# B&R Automation Studio project IP001 (part 2)

#### FValve.st
```iecst
(* ЗАДВИЖКА *)
FUNCTION_BLOCK FValve
	IF r0.14 THEN
		r0.14 := 0;
		Failures := 0;
	END_IF
	IF Failures = 0 THEN					//Сброс таймаутов
		TimeoutC := 0;
		TimeoutO := 0;
		OpenNoAllow := 0;
		CloseNoAllow := 0;
		NoOpenNoAllow := 0;
		NoCloseNoAllow := 0;
	END_IF;
	(* разбираем регистр команд *)
	IF r0.0 THEN
		Open := 1;	r0.0 := 0;
	END_IF;
	IF r0.1 THEN
		Close := 1;	r0.1 := 0;
	END_IF;
	IF r0.2 THEN
		Stop := 1; r0.2 := 0;
	END_IF

	Block	:= r0.3;
	Auto	:= r0.5;
	Imitation := r0.13;

	IF PAZ THEN
		Open := 0;
		Close := 0;
		Stop := 0;
	END_IF
	(* Блокировка неактуальных команд *)
	IF Block THEN
		Open	:= 0;
		Close	:= 0;
		Stop	:= 0;
	END_IF;

	IF Open AND Opened THEN
		Open := 0;
	END_IF;
	IF Close AND Closed THEN
		Close := 0;
	END_IF;
	(*	режим иммитации	*)
	IF NOT Imitation THEN
		Opened	:= OpenedDI;
		Closed	:= ClosedDI;
	ELSE
		IF Opening AND T.ET > T#2s THEN Opened	:= 1; END_IF;
		IF Closing AND T.ET > T#2s THEN Closed	:= 1; END_IF;
	END_IF;
	(* команды *)
	IF Open THEN									// команда ОТКРЫТЬ
		Closing	:= 0;
		Closed	:= 0;
		CloseDO	:= 0;
		Open	:= 0;
		Opening	:= 1;
		OpenDO	:= 1 AND NOT Imitation AND NOT PAZ;
		T(IN	:= 1);
	END_IF;
	IF Opening AND Opened THEN						// Открылась
		Opening	:= 0;
		OpenDO	:= 0;
		OpenDIOld := OpenedDI;
		StopDO	:= 1  AND NOT Imitation;
		T(IN	:= 0);
	END_IF;
	IF Opening AND T.Q THEN							// НЕ Открылась
		Opening	:= 0;
		OpenDO	:= 0;
		T(IN	:= 0);
		TimeoutO:= 1;
	END_IF;

	IF Close THEN											// команда ЗАКРЫТЬ
		Opening	:= 0;
		Opened	:= 0;
		OpenDO	:= 0;
		Close	:= 0;
		Closing	:= 1;
		CloseDO	:= 1 AND NOT Imitation AND NOT PAZ;
		T(IN	:= 1);
	END_IF;
	IF Closing AND Closed THEN								// Закрылась
		Closing	:= 0;
		CloseDO	:= 0;
		CloseDIOld := ClosedDI;
		T(IN	:= 0);
		StopDO	:= 1;
	END_IF;
	IF Closing AND T.Q THEN									// НЕ Закрылась
		Closing	:= 0;
		CloseDO	:= 0;
		T(IN	:= 0);
		TimeoutC:= 1;
	END_IF;

	IF Stop	THEN											// Команда СТОП
		Stop	:= 0;
		Opening	:= 0;
		Closing	:= 0;
		OpenDO	:= 0;
		CloseDO	:= 0;
		T.IN	:= 0;
		StopDO	:= 1 AND NOT Imitation AND NOT PAZ;
	END_IF;

	IF StopPresent AND TSignal.Q THEN						// DO сигналы делаем 1 сек если есть сигнал StopDO
		OpenDO	:= 0;
		CloseDO	:= 0;
		StopDO	:= 0;
	END_IF;

	IF Block THEN											// при блокеровке обнуляем выходные сигналы
		OpenDO	:= 0;
		CloseDO	:= 0;
		StopDO	:= 0;
	END_IF;
	// Блокировка по ПАЗ или команда РЕМОНТ
	IF PAZ OR r0.10 THEN
		Opening	:= 0;
		Closing	:= 0;
		OpenDO	:= 0;
		CloseDO	:= 0;
		T.IN	:= 0;
		StopDO	:= 0;
	END_IF;
	(* Самопроизвольное открытие/закрытие *)
	IF Opening AND NOT ClosedDI THEN
		CloseDIOld := 0;
	END_IF;
	IF Closing AND NOT OpenedDI THEN
		OpenDIOld := 0;
	END_IF;
	IF OpenedDI AND NOT OpenDIOld THEN
		OpenDIOld := OpenedDI;
		OpenNoAllow := 1;
	END_IF;
	IF ClosedDI AND NOT CloseDIOld THEN
		CloseDIOld := ClosedDI;
		CloseNoAllow := 1;
	END_IF;
	IF NOT OpenedDI AND OpenDIOld THEN
		OpenDIOld := OpenedDI;
		NoOpenNoAllow := 1;
	END_IF;
	IF NOT ClosedDI AND CloseDIOld THEN
		CloseDIOld := ClosedDI;
		NoCloseNoAllow := 1;
	END_IF;
	(* Утечки *)
	// LeakTON(IN := LeakDI, PT := DINT_TO_TIME(LeakageTimer));
	// вызов таймера хода (30 сек по дефолту)
	T(PT := DINT_TO_TIME(FullTimerInterval));
	TSignal(IN := CloseDO OR OpenDO OR StopDO);
	(* Регистр состояний *)
	r1.0	:= NOT Block;									//  программный 1:может управл с контроллера; 0:только слежение за состоянием, без управл
	r1.1	:= TimeoutC OR TimeoutO;									// контроль (наличие) протечки
	r1.2	:= Auto;										// Режим АВТОМАТИЧЕСКИЙ
	r1.3 	:= NOT Auto;									// Режим РУЧНОЙ
	r1.4	:= Opening;										//  открывается
	r1.5	:= Closing;										//  закрывается
	r1.6	:= Opened;										//	открыта
	r1.7	:= Closed;										//	закрыта
	r1.8	:= (NOT OpenedDI AND NOT ClosedDI)AND NOT(OpenDO OR CloseDO);					//	в промежуточном положении

	//r1.10	:= AlarmDI;										// аварийное отключение или сработала муфта
	//r1.11 связи с интерфейсной задвижкой (0-нет связи, 1-есть связь)
	r1.12	:= NOT Block;									//	Работоспособен:= (если программный или имитационный, и если не блокирован)
	r1.13	:= NOT Block AND NOT PAZ AND NOT r0.10;		//	Готова
	r1.14	:= PAZ;											// задвижка под управлением ПАЗ
	(* Регистор аварий *)
	Failures.0	:= TimeoutC OR TimeoutO;					// Не открылась/закрылась за время T.PT
	// превышение времени схода с концевого выключателя
	Failures.2	:= TimeoutC OR TimeoutO;					// превышение времени полного хода вала
	// 3
	Failures.4	:= TimeoutO;								//	не выполнение команды открыть
	Failures.5	:= TimeoutC;								//	не выполнение команды закрыть
	// 6
	//7	сработала электрозащита
	//8	невыполнение команды останова
	//9	Сработал моментный выключатель открытия
	//10	Сработал моментный выключатель закрытия
	//11	Привод перегрелся
	Failures.12 := OpenNoAllow;
	Failures.13 := CloseNoAllow;
	Failures.14 := NoOpenNoAllow;
	Failures.15 := NoCloseNoAllow;

END_FUNCTION_BLOCK
```

#### FAI.st
```iecst
(* Обработка AI *)
FUNCTION_BLOCK FAI
	ImitationEn := 	RegCmd.1;
	HiEnabled := 	RegCmd.4;
	HiHiEnabled :=	RegCmd.5;
	LoEnabled := 	RegCmd.6;
	LoLoEnabled := 	RegCmd.7;
	Scale := HiScale - LoScale;	//шкала
	CASE ChannelType OF
		0:
			Current := RAW*20.0/32767.0;
			Value := RAW*((Scale+Scale/4)/32767.0) + (LoScale - Scale/4.0);
			Invalid := (ChannelOverflow OR ChannelUnderflow OR Current <= 3.2) AND NOT ImitationEn;// КЗ/обрыв
		1:
			Current := RAW*16.0/32767.0 + 4.0;
			Value := RAW*(Scale /32767.0) + LoScale;
			Invalid := (ChannelOverflow OR ChannelUnderflow OR Current <= 3.2) AND NOT ImitationEn;// КЗ/обрыв
		2:
			Current := RAW*22.0/32767.0;
			Value := RAW*(Scale+Scale/4)/32767.0 - Scale/4;
			Invalid := (ChannelOverflow OR ChannelUnderflow) AND NOT ImitationEn;// КЗ/обрыв
		3:
			Current := 0;
			Value := MbValue;
			Invalid := (ChannelOverflow OR ChannelUnderflow) AND NOT ImitationEn;// КЗ/обрыв
	END_CASE
	//Value := (Current - 4.0) / 16.0 * Scale + LoScale;
	IF ImitationEn THEN
		Value := Replace_Value;	// подстановочное
	ELSE
		IF Value < LoScale THEN
			Value := LoScale;
		END_IF;
		IF Value > HiScale THEN
			Value := HiScale;
		END_IF;
	END_IF;

	(* Аварии *)
	IF LoLoAlarm AND (Value >= (LoLoLimit + Scale*(Hyst/100.0)))OR  NOT LoLoEnabled OR Invalid THEN
		LoLoAlarm := 0;
	END_IF;
	IF NOT LoLoAlarm AND (Value < LoLoLimit)AND LoLoEnabled AND NOT Invalid THEN
		LoLoAlarm := 1;
	END_IF;
	IF LoAlarm AND (Value >= (LoLimit + Scale*(Hyst/100.0)))OR  NOT LoEnabled OR Invalid THEN
		LoAlarm := 0;
	END_IF;
	IF NOT LoAlarm AND (Value < LoLimit)AND LoEnabled AND NOT Invalid THEN
		LoAlarm := 1;
	END_IF;
	IF HiAlarm AND (Value <= (HiLimit - Scale*(Hyst/100.0)))OR  NOT HiEnabled OR Invalid THEN
		HiAlarm := 0;
	END_IF;
	IF NOT HiAlarm AND (Value > HiLimit)AND HiEnabled AND NOT Invalid THEN
		HiAlarm := 1;
	END_IF;
	IF HiHiAlarm AND (Value <= (HiHiLimit - Scale*(Hyst/100.0)))OR  NOT HiHiEnabled OR Invalid THEN
		HiHiAlarm := 0;
	END_IF;
	IF NOT HiHiAlarm AND (Value > HiHiLimit )AND HiHiEnabled AND NOT Invalid THEN
		HiHiAlarm := 1;
	END_IF;

	Color := 1;
	IF LoAlarm OR HiAlarm THEN
		Color := 2;
	END_IF
	IF LoLoAlarm OR HiHiAlarm THEN
		Color := 3;
	END_IF
	IF Invalid THEN
		Color := 4;
	END_IF

	RegStatus.0	:= Invalid;						//Сигнал достоверен (=FALSE) или нет (=TRUE)
	RegStatus.1	:= HiAlarm;						//Значение выше чем предупредительная уставка "HiLimit"
	RegStatus.2	:= HiHiAlarm;					//Значение выше чем аварийная уставка "HiHiLimit"
	RegStatus.3	:= LoAlarm;						//Значение ниже чем предупредительная уставка "LoLimit"
	RegStatus.4	:= LoLoAlarm;					//Значение ниже чем аварийная уставка "LoLoLimit"
	RegStatus.5 := ImitationEn;					//Включена имитация

END_FUNCTION_BLOCK
```

#### FDI.st
```iecst
(*Обработка дискретных входов*)
FUNCTION_BLOCK FDI
	Out := ((In XOR Inv) AND NOT MaskEn)OR(MaskEn AND Mask);
END_FUNCTION_BLOCK
```

#### FDO.st
```iecst
(*Обработка дискретных выходов*)
FUNCTION_BLOCK FDO
	Out	:= ((In	XOR Inv)	AND NOT MaskEn)	OR(MaskEn		AND Mask);
END_FUNCTION_BLOCK
```

#### FAO.st
```iecst
(* Обработка AO *)
FUNCTION_BLOCK FAO

	Scale := HiScale - LoScale;										//шкала
	IF ImitationEn THEN
		Value := Replace_Value;	  									// подстановочное
	END_IF

	RAW := REAL_TO_INT((Value-LoScale)*(32767.0)/(HiScale-LoScale));		// Величину в АЦП канала
	Current := RAW*16.0/32767.0+4.0;										// АЦП в ТОК

	(* Аварии *)
	IF LoLoAlarm AND (Value > (LoLoLimit + Scale/200.0))OR  NOT LoLoEnabled OR Invalid THEN
		LoLoAlarm := 0;
	END_IF;
	IF NOT LoLoAlarm AND (Value < (LoLoLimit - Scale/200.0))AND LoLoEnabled AND NOT Invalid THEN
		LoLoAlarm := 1;
	END_IF;
	IF LoAlarm AND (Value > (LoLimit + Scale/200.0))OR  NOT LoEnabled OR Invalid THEN
		LoAlarm := 0;
	END_IF;
	IF NOT LoAlarm AND (Value < (LoLimit - Scale/200.0))AND LoEnabled AND NOT Invalid THEN
		LoAlarm := 1;
	END_IF;
	IF HiAlarm AND (Value < (HiLimit - Scale/200.0))OR  NOT HiEnabled OR Invalid THEN
		HiAlarm := 0;
	END_IF;
	IF NOT HiAlarm AND (Value > (HiLimit + Scale/200.0))AND HiEnabled AND NOT Invalid THEN
		HiAlarm := 1;
	END_IF;
	IF HiHiAlarm AND (Value < (HiHiLimit - Scale/200.0))OR  NOT HiHiEnabled OR Invalid THEN
		HiHiAlarm := 0;
	END_IF;
	IF NOT HiHiAlarm AND (Value > (HiHiLimit + Scale/200.0))AND HiHiEnabled AND NOT Invalid THEN
		HiHiAlarm := 1;
	END_IF;
END_FUNCTION_BLOCK
```

#### FPIDreg_r.st
```iecst
FUNCTION_BLOCK FPIDreg_r
	IF AlOpen THEN mode := 3; END_IF
	IF AlClose THEN mode := 4; END_IF
	IF enable THEN
		status := 0;
		MTBasicsPID_0.Invert := invert;
		MTBasicsPID_0.MinOut := Y_min;
		MTBasicsPID_0.MaxOut := Y_max;
		MTBasicsPID_0.SetValue := X_set;
		MTBasicsPID_0.ActValue := X;
		IF (MTBasicsPID_0.PIDParameters.Gain <> Gain) OR (MTBasicsPID_0.PIDParameters.IntegrationTime <> IntegrationTime)
			OR (MTBasicsPID_0.PIDParameters.DerivativeTime <> DerivativeTime)OR (MTBasicsPID_0.PIDParameters.FilterTime <> FilterTime) THEN
			MTBasicsPID_0.PIDParameters.Gain := Gain;
			MTBasicsPID_0.PIDParameters.IntegrationTime := IntegrationTime;
			MTBasicsPID_0.PIDParameters.DerivativeTime := DerivativeTime;
			MTBasicsPID_0.PIDParameters.FilterTime := FilterTime;
			MTBasicsPID_0.Update := TRUE;
		ELSE MTBasicsPID_0.Update := FALSE;
		END_IF
		CASE mode OF
			0://выключен
				MTBasicsPID_0.Enable := FALSE;
			1://автоматический режим
				MTBasicsPID_0.Enable := TRUE;
				MTBasicsPID_0.EnableTracking := FALSE;
				IF MTBasicsPID_0.IntegrationPartPresetValue <> MTBasicsPID_0.TrackingValue THEN
					MTBasicsPID_0.IntegrationPartPresetValue := MTBasicsPID_0.TrackingValue;
				END_IF
				IF NOT MTBasicsPID_0.EnableTracking AND MTBasicsPID_0.TrackingActive THEN
					MTBasicsPID_0.SetIntegrationPart := TRUE;
				ELSE 	MTBasicsPID_0.SetIntegrationPart := FALSE;
				END_IF
			2://ручной режим
				MTBasicsPID_0.Enable := TRUE;
				MTBasicsPID_0.EnableTracking := TRUE;
				MTBasicsPID_0.TrackingValue := Y_man;
			3://в ручном на макс
				MTBasicsPID_0.Enable := TRUE;
				MTBasicsPID_0.EnableTracking := TRUE;
				MTBasicsPID_0.TrackingValue := MTBasicsPID_0.MaxOut;
			4://в ручном на мин
				MTBasicsPID_0.Enable := TRUE;
				MTBasicsPID_0.EnableTracking := TRUE;
				MTBasicsPID_0.TrackingValue := MTBasicsPID_0.MinOut;
			ELSE
				mode := 2;
		END_CASE

		MTBasicsPID_0();
		Y_out := MTBasicsPID_0.Out;
		status := MTBasicsPID_0.StatusID;
	END_IF
END_FUNCTION_BLOCK
```

#### FMotor.st
```iecst
FUNCTION_BLOCK FMotor
	IF Block THEN
		Start	:= 0;
		Stop	:= 1;
	END_IF
	Started_old := Started;
	Stopped_old := Stopped;
	IF Block AND Started THEN
		Status.5 := TRUE;
	END_IF
	IF Status.5 AND Reset AND Stopped THEN
		Status.5 := FALSE;
	END_IF
	//Имитация
	IF NOT Imitation THEN
		Started := RunDI;
		Stopped := NOT RunDI;
	ELSE
		IF Start THEN Started := 1; Stopped := 0; END_IF
		IF Stop THEN Started := 0; Stopped := 1; END_IF
	END_IF
	IF Start AND Started THEN				// Блокировка неактуальных команд
		Start := 0;
	END_IF
	IF Stop AND Stopped THEN
		Stop := 0;
	END_IF
	IF Reset THEN							// Таймаут Сбрс
		Reset	:= 0;
		Timeout	:= 0;
	END_IF
	IF Start THEN							// СТАРТ
		Start	:= 0;
		StartDO	:= 1;
		T.IN := 1;
	END_IF
	IF Stop THEN							// СТОП
		Stop	:= 0;
		StopDO	:= 1;
		T.IN := 1;
	END_IF
	IF (StartDO OR StopDO) AND T.Q THEN		// Таймаут
		StartDO	:= 0;
		StopDO	:= 0;
		T.IN	:= 0;
		Timeout	:= 1;
	END_IF
	IF StartDO AND RunDI THEN				// Стартовал
		StartDO := 0;
		T.IN	:= 0;
		Timeout	:= 0;
	END_IF

	IF StopDO AND NOT RunDI THEN			// Остановился
		StopDO := 0;
		T.IN	:= 0;
		Timeout	:= 0;
	END_IF
	T(IN := T.IN,	PT := T#3s00ms);
	MH(Run := Started,Reset := ResetMH);
	ResetMH := 0;
	MotoHours := MH.Counter;
	Status.0	:= Started;
	Status.1 	:= Stopped;
	Status.2 	:= Block;
	Status.3	:= Timeout;
	Status.4	:= Timeout;

END_FUNCTION_BLOCK
```

#### PassportValve.st
```iecst
(* TODO: Add your comment here *)
FUNCTION_BLOCK PassportValve
	IF is_first THEN
		is_first := 0;
		cmdOpen := Gate_buf.r0.0;
		cmdClose := Gate_buf.r0.1;
		cmdBlck := Gate_buf.r0.3;
		cmdAuto := Gate_buf.r0.5;
		cmdImit := Gate_buf.r0.13;
		statePLC_control := Gate_buf.r1.0;
		stateLeak := Gate_buf.r1.1;
		stateAuto := Gate_buf.r1.2;
		stateManu := Gate_buf.r1.3;
		stateOpening := Gate_buf.r1.4;
		stateClosing := Gate_buf.r1.5;
		stateOpened := Gate_buf.r1.6;
		stateClosed := Gate_buf.r1.7;
		statePAZ := Gate_buf.r1.14;
		failTimeout := Gate_buf.Failures.0 OR Gate_buf.Failures.2;
		failTimeoutO := Gate_buf.Failures.4;
		failTimeoutC := Gate_buf.Failures.5;
		timePT := Gate_buf.FullTimerInterval/1000;
	ELSE
		Gate_buf.r0.0 := cmdOpen;
		Gate_buf.r0.1 := cmdClose;
		Gate_buf.r0.3 := cmdBlck;
		Gate_buf.r0.5 := cmdAuto;
		Gate_buf.r0.13 := cmdImit;
		statePLC_control := Gate_buf.r1.0;
		stateLeak := Gate_buf.r1.1;
		stateAuto := Gate_buf.r1.2;
		stateManu := Gate_buf.r1.3;
		stateOpening := Gate_buf.r1.4;
		stateClosing := Gate_buf.r1.5;
		stateOpened := Gate_buf.r1.6;
		stateClosed := Gate_buf.r1.7;
		statePAZ := Gate_buf.r1.14;
		failTimeout := Gate_buf.Failures.0 OR Gate_buf.Failures.2;
		failTimeoutO := Gate_buf.Failures.4;
		failTimeoutC := Gate_buf.Failures.5;
		Gate_buf.FullTimerInterval := timePT*1000;
		IF cmdResetAlarms THEN
			Gate_buf.r0.14 := 1;
			cmdResetAlarms := 0;
		END_IF
	END_IF
END_FUNCTION_BLOCK
```

#### PassportAI.st
```iecst
FUNCTION_BLOCK PassportAI
	IF is_first THEN
		index1_old	:= index1;
		index2_old	:= index2;
		is_first 	:= 0;
		LoScale 	:= AI_buf.LoScale;
		HiScale 	:= AI_buf.HiScale;
		HiLimit 	:= AI_buf.HiLimit;
		HiHiLimit 	:= AI_buf.HiHiLimit;
		LoLimit 	:= AI_buf.LoLimit;
		LoLoLimit 	:= AI_buf.LoLoLimit;
		current 	:= AI_buf.Current;
		Value 		:= AI_buf.Value;
		ImitVal 	:= AI_buf.Replace_Value;
		cmdImit 	:= AI_buf.ImitationEn;
		cmdHiEn 	:= AI_buf.HiEnabled;
		cmdHiHiEn 	:= AI_buf.HiHiEnabled;
		cmdLoEn 	:= AI_buf.LoEnabled;
		cmdLoLoEn 	:= AI_buf.LoLoEnabled;
		stateInvalid:= AI_buf.Invalid;
		stateHi 	:= AI_buf.HiAlarm;
		stateHiHi 	:= AI_buf.HiHiAlarm;
		stateLo 	:= AI_buf.LoAlarm;
		stateLoLo 	:= AI_buf.LoLoAlarm;

	ELSE
		IF index1_old = index1 AND index2_old = index2 THEN
			current := AI_buf.Current;
			Value := AI_buf.Value;
			stateInvalid:= AI_buf.Invalid;
			stateHi 	:= AI_buf.HiAlarm;
			stateHiHi 	:= AI_buf.HiHiAlarm;
			stateLo 	:= AI_buf.LoAlarm;
			stateLoLo 	:= AI_buf.LoLoAlarm;
			AI_buf.LoScale := LoScale;
			AI_buf.HiScale := HiScale;
			AI_buf.HiLimit := HiLimit;
			AI_buf.HiHiLimit := HiHiLimit;
			AI_buf.LoLimit := LoLimit;
			AI_buf.LoLoLimit := LoLoLimit;
			AI_buf.Replace_Value := ImitVal;
			AI_buf.ImitationEn := cmdImit;
			AI_buf.HiEnabled := cmdHiEn;
			AI_buf.HiHiEnabled := cmdHiHiEn;
			AI_buf.LoEnabled := cmdLoEn;
			AI_buf.LoLoEnabled := cmdLoLoEn;
		ELSE is_first := 1;
		END_IF
	END_IF

END_FUNCTION_BLOCK
```

#### FDISKRreg_r.st
```iecst
(* Дискретный регулятор *)
FUNCTION_BLOCK FDISKRreg_r
	IF enable THEN
		IF invert THEN //регулятор ПОСЛЕ СЕБЯ
			IF X < X_set_low 	THEN OnDO := TRUE; OffDO := FALSE; END_IF
			IF X > X_set_high THEN OnDO := FALSE; OffDO := TRUE; END_IF
		ELSE			//регулятор ДО СЕБЯ
			IF X > X_set_high THEN OnDO := TRUE; OffDO := FALSE; END_IF
			IF X < X_set_low 	THEN OnDO := FALSE; OffDO := TRUE; END_IF
		END_IF
	ELSE OnDO := FALSE; OffDO := TRUE;
	END_IF
END_FUNCTION_BLOCK
```

#### UVP_TCP.st
```iecst
(* UVP_TCP *)
FUNCTION_BLOCK UVP_TCP
	CASE step OF
		0://чтение текущего времени УВП(+маска описанных трубопроводов)
			req_3x (enable := TRUE,pStation := pPort,startAddress :=1800,nrRegisters :=SIZEOF(UVP_Data.Time)/2 ,pData := ADR(UVP_Data.Time),dataSize :=SIZEOF(UVP_Data.Time));
			IF req_3x.status <> ERR_FUB_BUSY THEN
				step := 1;
			END_IF
			state := req_3x.status;
		1://чтение порядка байт
			req_3x (enable := TRUE,pStation := pPort,startAddress :=100,nrRegisters :=SIZEOF(UVP_Data.Byte_order)/2 ,pData := ADR(UVP_Data.Byte_order),dataSize :=SIZEOF(UVP_Data.Byte_order));
			IF req_3x.status <> ERR_FUB_BUSY THEN
				step := 2;
			END_IF
			state := req_3x.status;
		2://запись порядка байт,если он отличается от заданного(#2301)
			IF UVP_Data.Byte_order <> UVP_Data.Byte_order_new THEN
				req_6x (enable := TRUE,pStation := pPort,startAddress :=100,value := UVP_Data.Byte_order_new);
				IF req_6x.status <> ERR_FUB_BUSY THEN
					step := 3;
				END_IF
				state := req_6x.status;
			ELSE step := 3;
			END_IF
		3://чтение текущих параметров трубопровода(за один проход CASE один трубопровод)
			WHILE ((curTP <= 15) AND ((UVP_Data.Time.TPs AND SHL(1,curTP)) = 0)) DO
				curTP := curTP + 1;
			END_WHILE
			IF curTP > 15 THEN curTP := 0; END_IF
			IF ((UVP_Data.Time.TPs AND SHL(1,curTP))<>0) THEN
				req_4x(enable := TRUE,pStation := pPort,startAddress := 2000+(curTP*100), nrRegisters := SIZEOF(UVP_Data.LineCurrent[curTP+1])/2,pData := ADR(UVP_Data.LineCurrent[curTP+1]),dataSize :=SIZEOF(UVP_Data.LineCurrent[curTP+1]));
				IF req_4x.status <> ERR_FUB_BUSY THEN
					step := 4;
				END_IF
				state := req_4x.status;
			ELSE step := 4;
			END_IF
			//чтение текущих архивов(за один проход CASE один трубопровод)
		4:	IF ((UVP_Data.Time.TPs AND SHL(1,curTP))<>0) THEN
				req_4x(enable := TRUE,pStation := pPort,startAddress := 2000+(curTP*100)+60, nrRegisters := SIZEOF(UVP_Data.Prev_hour[curTP+1])/2,pData := ADR(UVP_Data.Prev_hour[curTP+1]),dataSize :=SIZEOF(UVP_Data.Prev_hour[curTP+1]));
				IF req_4x.status <> ERR_FUB_BUSY THEN
					step := 5;
				END_IF
				state := req_4x.status;
			ELSE step := 5;
			END_IF
			//чтение текущих архивов(за один проход CASE один трубопровод)
		5:	IF ((UVP_Data.Time.TPs AND SHL(1,curTP))<>0) THEN
				req_4x (enable := TRUE,pStation := pPort,startAddress := 2000+(curTP*100)+80, nrRegisters := SIZEOF(UVP_Data.Prev_day[curTP+1])/2,pData := ADR(UVP_Data.Prev_day[curTP+1]),dataSize :=SIZEOF(UVP_Data.Prev_day[curTP+1]));
				IF req_4x.status <> ERR_FUB_BUSY THEN
					curTP := curTP + 1;
					step := 6;
				END_IF
				state := req_4x.status;
			ELSE step := 6;
			END_IF
		6:  //синхронизация времени  с NTP сервером(в конфиге контроллера включен сервер)
			//IP адрес контроллера задан младшим словом вперед,т.к. порядяок байт #2301
			IF UVP_Data.synchrooo THEN
				UVP_Data.synchrooo := FALSE;
				UVP_Data.NTP.IPAddr1 := UVP_Data.NTP.IpAddress3*256 + UVP_Data.NTP.IpAddress4;
				UVP_Data.NTP.IPAddr2 := UVP_Data.NTP.IpAddress1*256 + UVP_Data.NTP.IpAddress2;
				UVP_Data.NTP.cmd := 24680;
				req_16x(enable := TRUE,pStation := pPort, startAddress := 1005, nrRegisters := SIZEOF(UVP_Data.NTP)/2,pData:=ADR(UVP_Data.NTP),dataSize := SIZEOF(UVP_Data.NTP));
				IF req_16x.status <> ERR_FUB_BUSY THEN
					step := 7;
				END_IF
				state := req_16x.status;
			ELSE step := 7;
			END_IF
		7://чтение текущего статуса синхронизации времени
			req_3x (enable := TRUE,pStation := pPort, startAddress := 1005, nrRegisters := (SIZEOF(UVP_Data.NTP)-4)/2,pData:=ADR(UVP_Data.NTP),dataSize := SIZEOF(UVP_Data.NTP)-4);
			IF req_3x.status <> ERR_FUB_BUSY THEN
				step := 8;
			END_IF
			state := req_3x.status;
		8:
			req_3x (enable := TRUE,pStation := pPort, startAddress := 1008, nrRegisters := SIZEOF(UVP_Data.DeltaTime)/2,pData:=ADR(UVP_Data.DeltaTime),dataSize := SIZEOF(UVP_Data.DeltaTime));
			IF req_3x.status <> ERR_FUB_BUSY THEN
				step := 9;
			END_IF
			state := req_3x.status;
		9://чтение компонентного состава газовой смеси МР-113
			IF UVP_Data.read_gas_comp THEN
				req_3x(enable := TRUE,pStation := pPort, startAddress := 1100, nrRegisters := SIZEOF(UVP_Data.MR_113)/2,pData:=ADR(UVP_Data.MR_113),dataSize := SIZEOF(UVP_Data.MR_113));
				IF req_3x.status  <> ERR_FUB_BUSY THEN
					UVP_Data.MR_113_new := UVP_Data.MR_113;
					UVP_Data.read_gas_comp := FALSE;
					step := 10;
				END_IF
				state := req_3x.status;
			ELSE step := 10;
			END_IF
		10://запись компонентного состава газовой смеси МР-113
			IF UVP_Data.write_gas_comp THEN
				req_16x(enable := TRUE, pStation := pPort, startAddress := 1100, nrRegisters := SIZEOF(UVP_Data.MR_113_new)/2,pData:=ADR(UVP_Data.MR_113_new),dataSize := SIZEOF(UVP_Data.MR_113_new));
				IF req_16x.status <> ERR_FUB_BUSY THEN
					UVP_Data.write_gas_comp := FALSE;
					step := 0;
				END_IF
				state := req_16x.status;
			ELSE step := 0;
			END_IF
	END_CASE;

	IF state = 34201 THEN
			status := state;
			Timeout_T (IN := TRUE, PT := T#5000ms);
			IF Timeout_T.Q THEN
				step := step + 1;
				Timeout_T (IN := FALSE, PT := T#5000ms);
		END_IF
	ELSE status := 0;
	END_IF

	IF step > 10 THEN step := 0; END_IF
END_FUNCTION_BLOCK
```

#### FMHCounter.st
```iecst
(* FMHCounter *)
FUNCTION_BLOCK FMHCounter
	T(IN := Run, PT :=  UINT_TO_TIME(Tik*1000));
	IF T.Q THEN
		Counter := Counter + (Tik/3600.00);
		T(IN := FALSE);
	END_IF
	IF Reset THEN Counter := 0; END_IF
END_FUNCTION_BLOCK
```

#### FTorch.st
```iecst
(* Torch *)
FUNCTION_BLOCK FTorch
	Timer_vent(PT := UINT_TO_TIME(Time_vent*1000));
	Timer_firing(PT := UINT_TO_TIME(Time_firing*1000));
	Timer_stabiliz(PT := UINT_TO_TIME(Time_stabiliz*1000));
	Timer_spark_off(PT := UINT_TO_TIME(Time_spark_off*1000));
	Timer_spark_on(PT := UINT_TO_TIME(Time_spark_on*1000));
	Timer_after_alarm(PT := UINT_TO_TIME(Time_after_alarm*1000));

	IF Stop THEN
		Timer_vent.IN := FALSE;
		Timer_firing.IN := FALSE;
		Timer_stabiliz.IN := FALSE;
		Timer_spark_off.IN := FALSE;
		Timer_spark_on.IN := FALSE;
		Timer_after_alarm.IN := FALSE;
		Do_Valve := FALSE;
		Do_Spark := FALSE;
		Do_Lamp_P_Zapal_low := FALSE;
		Do_Lamp_FireON := FALSE;
		Do_Lamp_Alarm := FALSE;
		step := 0;
		Stop := FALSE;
	END_IF
	Do_Lamp_Alarm := USINT_TO_BOOL(Alarm);
	Do_Lamp_FireON := Di_Fire;
	IF NOT Mode_Manual THEN
		CASE step OF
			0://Начальное состояние(ГОТОВНОСТЬ К ПУСКУ)
				IF Di_Fire THEN Warning_2 := TRUE;
				ELSE Warning_2 := FALSE; END_IF;
				IF Di_P_gas_low THEN Warning_1 := TRUE;
				ELSE Warning_1 := FALSE; END_IF;
				IF Start AND NOT Di_Fire AND NOT Di_P_gas_low THEN
					Start := FALSE;
					step := 1;
					Alarm := 0;
					firing_count := 0;
				END_IF;
			1:// ВЕНТИЛЯЦИЯ
				IF NOT Di_P_gas_low THEN
					Do_Valve := TRUE;
					Timer_vent.IN := TRUE;
					IF Timer_vent.Q THEN
						Timer_vent.IN := FALSE;
						step := 2;
					END_IF;
				ELSE
					Do_Lamp_P_Zapal_low := TRUE;
					Do_Valve := FALSE;
					Timer_vent.IN := FALSE;
					step := 0;
					Alarm := 1;//Падение давления во время вентиляции
				END_IF;
			2://РОЗЖИГ
				IF NOT Di_P_gas_low THEN
					Timer_firing.IN := TRUE;
					Timer_spark_on.IN := NOT Timer_spark_off.Q;
					Timer_spark_off.IN := Timer_spark_on.Q;
					Do_Spark := NOT Timer_spark_on.Q;
					IF Di_Fire THEN
						Timer_firing.IN := FALSE;
						Timer_spark_on.IN := FALSE;
						Timer_spark_off.IN := FALSE;
						Do_Spark :=FALSE;
						step := 4;
					END_IF;
					IF Timer_firing.Q THEN
						Timer_firing.IN := FALSE;
						Timer_spark_on.IN := FALSE;
						Timer_spark_off.IN := FALSE;
						Do_Spark :=FALSE;
						step := 3;
					END_IF;
				ELSE
					Do_Lamp_P_Zapal_low := TRUE;
					Timer_firing.IN := FALSE;
					Timer_spark_on.IN := FALSE;
					Timer_spark_off.IN := FALSE;
					Do_Spark :=FALSE;
					Do_Valve := FALSE;
					step := 0;
					Alarm := 2;//Падение давления во время розжига
				END_IF

			3://СТАБИЛИЗАЦИЯ
				IF NOT Di_P_gas_low THEN
					Timer_stabiliz.IN := TRUE;
					IF Di_Fire THEN
						Timer_stabiliz.IN := FALSE;
						step := 4;
						Alarm := 0;
					END_IF;
					IF Timer_stabiliz.Q THEN
						Timer_stabiliz.IN := FALSE;
						step := 5;
						Alarm := 3; //Нет розжига
					END_IF;
				ELSE
					Timer_stabiliz.IN := FALSE;
					Do_Lamp_P_Zapal_low := TRUE;
					Do_Valve := FALSE;
					step := 0;
					Alarm := 4;//Падение давления во время стабилизации
				END_IF
			4://ГОРЕНИЕ
				IF Di_P_gas_low THEN
					Alarm := 6;//Падение давления во время горения
					step := 5;
					Do_Lamp_P_Zapal_low := TRUE;
				END_IF
				IF NOT Di_Fire THEN
					Alarm := 7; //Срыв пламени
					firing_count := firing_count + 1;
					IF firing_count > 3 THEN
						step := 0;
					ELSE
						step := 2;
					END_IF
				END_IF
			5://АВАРИЯ
				Do_Valve := FALSE;
				Timer_after_alarm.IN := TRUE;
				IF Timer_after_alarm.Q THEN
					Timer_after_alarm.IN := FALSE;
					step := 0;
				END_IF
		END_CASE
	END_IF
END_FUNCTION_BLOCK
```

#### ABAK_TCP.st
```iecst
(* ABAK_MB_TCP *)
FUNCTION_BLOCK ABAK_TCP
	CASE step OF
		0:
		1:
		2:
		3:
		4:
	END_CASE
END_FUNCTION_BLOCK
```

#### FSwitch.st
```iecst
(* Switch *)
FUNCTION_BLOCK FSwitch
	IF Block THEN
		Start_1	:= 0;
		Start_2	:= 0;
		Stop	:= 1;
	END_IF
	IF Block_1 THEN
		Start_1 := 0;
	END_IF
	IF Block_2 THEN
		Start_2 := 0;
	END_IF
	IF Block_Stop THEN
		Stop := 0;
	END_IF
	//Имитация
	IF NOT Imitation THEN
		Started_1 := RunDI_1;
		Started_2 := RunDI_2;
		Stopped := NOT (RunDI_1 OR RunDI_2);
	ELSE
		IF Start_1 THEN Started_1 := 1; Started_2 := 0; Stopped := 0; END_IF
		IF Start_2 THEN Started_2 := 1; Started_1 := 0; Stopped := 0; END_IF
		IF Stop THEN Started_1 := 0; Started_2 := 0; Stopped := 1; END_IF
	END_IF

	IF Start_1 AND Started_1 THEN				// Блокировка неактуальных команд
		Start_1 := 0;
	END_IF
	IF Start_2 AND Started_2 THEN				// Блокировка неактуальных команд
		Start_2 := 0;
	END_IF
	IF Stop AND Stopped THEN
		Stop := 0;
	END_IF
	IF Reset THEN							// Таймаут Сбрс
		Reset	:= 0;
		Timeout	:= 0;
	END_IF
	IF Start_1 THEN							// СТАРТ
		Start_1	:= 0;
		Starting_1 := 1;
		Stop := 1;
	END_IF
	IF Start_2 THEN							// СТАРТ
		Start_2	:= 0;
		Starting_2 := 1;
		Stop := 1;
	END_IF
	IF Starting_1 AND Stopped THEN
		Starting_1 := 0;
		StartDO_1 := 1;
		T.IN := 1;
	END_IF
	IF Starting_2 AND Stopped THEN
		Starting_2 := 0;
		StartDO_2 := 1;
		T.IN := 1;
	END_IF
	IF Stop THEN							// СТОП
		Stop	:= 0;
		StopDO	:= 1;
		T.IN := 1;
	END_IF
	IF (StartDO_1 OR StartDO_2 OR StopDO) AND T.Q THEN		// Таймаут
		StartDO_1	:= 0;
		StartDO_2	:= 0;
		StopDO	:= 0;
		T.IN	:= 0;
		Timeout	:= 1;
	END_IF
	IF StartDO_1 AND RunDI_1 THEN				// Стартовал
		StartDO_1 := 0;
		T.IN	:= 0;
		Timeout	:= 0;
	END_IF
	IF StartDO_2 AND RunDI_2 THEN				// Стартовал
		StartDO_2 := 0;
		T.IN	:= 0;
		Timeout	:= 0;
	END_IF
	IF StopDO AND NOT RunDI_1 AND NOT RunDI_2 THEN			// Остановился
		StopDO := 0;
		T.IN	:= 0;
		Timeout	:= 0;
	END_IF
	T(IN := T.IN,	PT := T#3s00ms);

	Status.0	:= Started_1;
	Status.1	:= Started_2;
	Status.2 	:= Stopped;
	Status.3	:= Timeout;
	Status.4 	:= Block_1;
	Status.5 	:= Block_2;
	Status.6  	:= Block_Stop;

END_FUNCTION_BLOCK
```

#### fCmdCOM.st
```iecst
(* MBRTU Comm to ATV *)
FUNCTION_BLOCK fCmdCOM
	MBMCmd_0.ident := ident;
	MBMCmd_0.mfc := cmd;
	MBMCmd_0.node := node;
	MBMCmd_0.offset := offset;
	MBMCmd_0.len := length;
	MBMCmd_0.data := pData;
	MBMCmd_0(enable := TRUE);
	status := MBMCmd_0.status;
END_FUNCTION_BLOCK
```

#### fOpenCOM.st
```iecst
(*  *)
FUNCTION_BLOCK fOpenCOM
	IF enable THEN
		MBMOpen_0(enable := TRUE, pDevice := Device, pMode := Mode, pConfig := Config, timeout := 1500 );
		status := MBMOpen_0.status;
		ident := MBMOpen_0.ident;
		enable := FALSE;
	END_IF
END_FUNCTION_BLOCK
```

#### fCloseCOM.st
```iecst
(*  *)
FUNCTION_BLOCK fCloseCOM
	IF enable THEN
		MBMClose_0.ident := ident;
		MBMClose_0(enable := TRUE);
		status := MBMClose_0.status;
		enable := FALSE;
	END_IF
END_FUNCTION_BLOCK
```

#### FAlarm.st
```iecst
(* Alarm with delay *)
FUNCTION_BLOCK FAlarm
	Result := IN AND EN;
	IF Ack AND (Result = 0) THEN
		Timer(IN := FALSE);
		OUT := FALSE;
		OUT_int := Result;
	END_IF

	Timer(IN := UINT_TO_BOOL(Result), PT := UINT_TO_TIME(Delay*1000));
	IF Timer.Q THEN
		OUT := TRUE;
		OUT_int := Result;
	END_IF
END_FUNCTION_BLOCK
```

#### UVP_RTU.st
```iecst
(* UVP over RTU *)
FUNCTION_BLOCK UVP_RTU
	CASE step OF
			0://чтение текущего времени УВП(+маска описанных трубопроводов)
				req_3x (enable := TRUE,pStation := pPort,startAddress :=1800,nrRegisters :=SIZEOF(UVP_Data.Time)/2 ,pData := ADR(UVP_Data.Time),dataSize :=SIZEOF(UVP_Data.Time));
				IF req_3x.status <> ERR_FUB_BUSY THEN
					step := 1;
				END_IF
				state := req_3x.status;
			1://чтение порядка байт
				req_3x (enable := TRUE,pStation := pPort,startAddress :=100,nrRegisters :=SIZEOF(UVP_Data.Byte_order)/2 ,pData := ADR(UVP_Data.Byte_order),dataSize :=SIZEOF(UVP_Data.Byte_order));
				IF req_3x.status <> ERR_FUB_BUSY THEN
					step := 2;
				END_IF
				state := req_3x.status;
			2://запись порядка байт,если он отличается от заданного(#2301)
				IF UVP_Data.Byte_order <> UVP_Data.Byte_order_new THEN
					req_6x (enable := TRUE,pStation := pPort,startAddress :=100,pData := ADR(UVP_Data.Byte_order_new));
					IF req_6x.status <> ERR_FUB_BUSY THEN
						step := 3;
					END_IF
					state := req_6x.status;
				ELSE step := 3;
				END_IF
			3://чтение текущих параметров трубопровода(за один проход CASE один трубопровод)
				WHILE ((curTP <= 15) AND ((UVP_Data.Time.TPs AND SHL(1,curTP)) = 0)) DO
					curTP := curTP + 1;
				END_WHILE
				IF curTP > 15 THEN curTP := 0; END_IF
				IF ((UVP_Data.Time.TPs AND SHL(1,curTP))<>0) THEN
					req_4x(enable := TRUE,pStation := pPort,startAddress := 2000+(curTP*100), nrRegisters := SIZEOF(UVP_Data.LineCurrent[curTP+1])/2,pData := ADR(UVP_Data.LineCurrent[curTP+1]),dataSize :=SIZEOF(UVP_Data.LineCurrent[curTP+1]));
					IF req_4x.status <> ERR_FUB_BUSY THEN
						step := 4;
					END_IF
					state := req_4x.status;
				ELSE step := 4;
				END_IF
				//чтение текущих архивов(за один проход CASE один трубопровод)
			4:	IF ((UVP_Data.Time.TPs AND SHL(1,curTP))<>0) THEN
					req_4x(enable := TRUE,pStation := pPort,startAddress := 2000+(curTP*100)+60, nrRegisters := SIZEOF(UVP_Data.Prev_hour[curTP+1])/2,pData := ADR(UVP_Data.Prev_hour[curTP+1]),dataSize :=SIZEOF(UVP_Data.Prev_hour[curTP+1]));
					IF req_4x.status <> ERR_FUB_BUSY THEN
						step := 5;
					END_IF
					state := req_4x.status;
				ELSE step := 5;
				END_IF
				//чтение текущих архивов(за один проход CASE один трубопровод)
			5:	IF ((UVP_Data.Time.TPs AND SHL(1,curTP))<>0) THEN
					req_4x (enable := TRUE,pStation := pPort,startAddress := 2000+(curTP*100)+80, nrRegisters := SIZEOF(UVP_Data.Prev_day[curTP+1])/2,pData := ADR(UVP_Data.Prev_day[curTP+1]),dataSize :=SIZEOF(UVP_Data.Prev_day[curTP+1]));
					IF req_4x.status <> ERR_FUB_BUSY THEN
						curTP := curTP + 1;
						step := 6;
					END_IF
					state := req_4x.status;
				ELSE step := 6;
				END_IF
			6:  //синхронизация времени  с NTP сервером(в конфиге контроллера включен сервер)
				//IP адрес контроллера задан младшим словом вперед,т.к. порядяок байт #2301
				IF UVP_Data.synchrooo THEN
					UVP_Data.synchrooo := FALSE;
					UVP_Data.NTP.IPAddr1 := UVP_Data.NTP.IpAddress3*256 + UVP_Data.NTP.IpAddress4;
					UVP_Data.NTP.IPAddr2 := UVP_Data.NTP.IpAddress1*256 + UVP_Data.NTP.IpAddress2;
					UVP_Data.NTP.cmd := 24680;
					req_16x(enable := TRUE,pStation := pPort, startAddress := 1005, nrRegisters := SIZEOF(UVP_Data.NTP)/2,pData:=ADR(UVP_Data.NTP),dataSize := SIZEOF(UVP_Data.NTP));
					IF req_16x.status <> ERR_FUB_BUSY THEN
						step := 7;
					END_IF
					state := req_16x.status;
				ELSE step := 7;
				END_IF
			7://чтение текущего статуса синхронизации времени
				req_3x (enable := TRUE,pStation := pPort, startAddress := 1005, nrRegisters := (SIZEOF(UVP_Data.NTP)-4)/2,pData:=ADR(UVP_Data.NTP),dataSize := SIZEOF(UVP_Data.NTP)-4);
				IF req_3x.status <> ERR_FUB_BUSY THEN
					step := 8;
				END_IF
				state := req_3x.status;
			8:
				req_3x(enable := TRUE,pStation := pPort, startAddress := 1008, nrRegisters := SIZEOF(UVP_Data.DeltaTime)/2,pData:=ADR(UVP_Data.DeltaTime),dataSize := SIZEOF(UVP_Data.DeltaTime));
				IF req_3x.status <> ERR_FUB_BUSY THEN
					step := 9;
				END_IF
				state := req_3x.status;
			9://чтение компонентного состава газовой смеси МР-113
				IF UVP_Data.read_gas_comp THEN
					req_3x(enable := TRUE,pStation := pPort, startAddress := 1100, nrRegisters := SIZEOF(UVP_Data.MR_113)/2,pData:=ADR(UVP_Data.MR_113),dataSize := SIZEOF(UVP_Data.MR_113));
					IF req_3x.status  <> ERR_FUB_BUSY THEN
						UVP_Data.MR_113_new := UVP_Data.MR_113;
						UVP_Data.read_gas_comp := FALSE;
						step := 10;
					END_IF
					state := req_3x.status;
				ELSE step := 10;
				END_IF
			10://запись компонентного состава газовой смеси МР-113
				IF UVP_Data.write_gas_comp THEN
					req_16x(enable := TRUE, pStation := pPort, startAddress := 1100, nrRegisters := SIZEOF(UVP_Data.MR_113_new)/2,pData:=ADR(UVP_Data.MR_113_new),dataSize := SIZEOF(UVP_Data.MR_113_new));
					IF req_16x.status <> ERR_FUB_BUSY THEN
						UVP_Data.write_gas_comp := FALSE;
						step := 0;
					END_IF
					state := req_16x.status;
				ELSE step := 0;
				END_IF
		END_CASE;

		IF state = 34201 THEN
			status := state;
			Timeout_T (IN := TRUE, PT := T#5000ms);
			IF Timeout_T.Q THEN
				step := step + 1;
				Timeout_T (IN := FALSE, PT := T#5000ms);
			END_IF
		ELSE status := 0;
		END_IF

		IF step > 10 THEN step := 0; END_IF
END_FUNCTION_BLOCK
```

#### mbReadHoldingRegs.st
```iecst
(*  *)
FUNCTION_BLOCK mbReadHoldingRegs
	CmdCOM(ident := pStation, cmd := 3, node := 1, pData := pData, offset := startAddress, length := nrRegisters);
END_FUNCTION_BLOCK
```

#### mbReadInputRegs.st
```iecst
(*  *)
FUNCTION_BLOCK mbReadInputRegs
	CmdCOM(ident := pStation, cmd := 4, node := 1, pData := pData, offset := startAddress, length := nrRegisters);
END_FUNCTION_BLOCK
```

#### mbWriteSingleReg.st
```iecst
(*  *)
FUNCTION_BLOCK mbWriteSingleReg
	CmdCOM(ident := pStation, cmd := 6, node := 1, pData := pData, offset := startAddress, length := nrRegisters);
END_FUNCTION_BLOCK
```

#### mbWriteMultipleRegs.st
```iecst
(*  *)
FUNCTION_BLOCK mbWriteMultipleRegs
	CmdCOM(ident := pStation, cmd := 16, node := 1, pData := pData, offset := startAddress, length := nrRegisters);
END_FUNCTION_BLOCK
```

#### ATV_Control.st
```iecst
(* Управление ПЧ через Модбас *)
FUNCTION_BLOCK ATV_Control
	IF  PortIdent <> 0 THEN
		//постоянно читаем параметры ПЧ
		CASE step OF
			0:
				CmdCOM(ident := PortIdent, mfc := 3, node := MB_Addr, offset := 3240, len := SIZEOF(HMIS)/2, data := ADR(HMIS));
				IF CmdCOM.status = 0 THEN
					step := 1;
					IF step_old = 2 THEN
						step := 3;
					END_IF
					IF HMIS = 3 THEN
						stStopped := TRUE;
					ELSE stStopped := FALSE;
					END_IF
					IF HMIS = 4 OR HMIS = 5 THEN
						stStarted := TRUE;
					ELSE stStarted := FALSE;
					END_IF
				END_IF
			1:	//пишем команду стоп
				IF cmdStop AND NOT stStopped THEN
					CMD := 0;
					CmdCOM(ident := PortIdent, mfc := 16, node := MB_Addr, offset := 8501, len := SIZEOF(CMD)/2, data := ADR(CMD));
					IF CmdCOM.status = 0 THEN
						step := 0;
							END_IF
				ELSE step := 2;
				END_IF
			2://пишем команду 6
				IF cmdStart AND NOT stStarted THEN
					CMD := 6;
					CmdCOM(ident := PortIdent, mfc := 16, node := MB_Addr, offset := 8501, len := SIZEOF(CMD)/2, data := ADR(CMD));
					IF CmdCOM.status = 0 THEN
						step := 0;
					END_IF
				ELSE step := 4;
				END_IF
			3://пишем команду 15
				IF HMIS = 2 THEN
					CMD := 15;
					CmdCOM(ident := PortIdent, mfc := 16, node := MB_Addr, offset := 8501, len := SIZEOF(CMD)/2, data := ADR(CMD));
					IF CmdCOM.status = 0 THEN
						step := 4;
					END_IF
				ELSE step := 4;
				END_IF
			4:
				CmdCOM(ident := PortIdent, mfc := 3, node := MB_Addr, offset := 3202, len := SIZEOF(RFR)/2, data := ADR(RFR));
				IF CmdCOM.status = 0 THEN
					OUT_Freq := RFR *  10.0;
					step := 5;
				END_IF
			5:
				LFR := REAL_TO_UINT(IN_Freq/10.0);
				CmdCOM(ident := PortIdent, mfc := 16, node := MB_Addr, offset := 8502, len := SIZEOF(LFR)/2, data := ADR(LFR));
				IF CmdCOM.status = 0 THEN
					step := 0;
				END_IF
			ELSE step := 0;
		END_CASE
		step_old := step;
	END_IF
END_FUNCTION_BLOCK
```

#### fAuma_MB.st
```iecst
(*  *)
FUNCTION_BLOCK fAuma_MB

	IF mode > 1 THEN mode := 0; END_IF

	CASE step OF
		0://чтенеи текущего состояние и положения
			CmdCOM(node := mbAddr, cmd := 4, offset := 1000,length := 3,pData := ADR(read), ident := identCOM);
			IF CmdCOM.status = 0 THEN
				curPosition := read.Pos/10.0;	//Положение
				state.0 := read.state_1.0; 		//Открыт
				state.1 := read.state_1.1;		//Закрыт
				state.3 := read.state_1.3;		//Местный
				state.4 := read.state_1.4;		//Открывается
				state.5 := read.state_1.5;		//Закрывается
				step := 1;
			END_IF

		1://в режиме задвижки
			IF mode = 0 THEN
				write.cmd := cmd AND 11;//убираем бит работы по уставке
				CmdCOM(node := mbAddr, cmd := 16, offset := 1000,length := 1,pData := ADR(write.cmd), ident := identCOM);
				IF CmdCOM.status = 0 THEN
					step := 0;
				END_IF
			ELSE
				step := 2;
			END_IF

		2://в режиме регулятора
			IF mode = 1 THEN
				write.Pos := REAL_TO_UINT(setPosition * 10);
				write.cmd := 4; //убираем все биты кроме бита работы по уставке
				CmdCOM(node := mbAddr, cmd := 16, offset := 1000,length := 2,pData := ADR(write), ident := identCOM);
				IF CmdCOM.status = 0 THEN
					step := 0;
				END_IF
			ELSE
				step := 1;
			END_IF

		ELSE step := 0;
	END_CASE

END_FUNCTION_BLOCK
```

### Library Logical/Libraries/LibIP001 (IEC)

#### Types.typ - Exported data types
```iecst
TYPE
	Biffi_Data : 	STRUCT
		Status : UINT;
		Cur_Position : UINT;
		Commands : UINT;
		Set_Position : UINT;
	END_STRUCT;
END_TYPE
```

#### Valve_Biffi.st
```iecst
(* Biffi valve modbus *)
(*
бит0-закрыть
бит1-открыть
бит2-стоп
бит4-управление положением
*)
FUNCTION_BLOCK Valve_Biffi
	(* Блокировка неактуальных команд *)
	IF r0.0 THEN//close
		IF r1.7 THEN// if closed
			r0.0 := 0;
		ELSE
			r0.1 := 0;
			r0.2 := 0;
		END_IF;
	END_IF;

	IF r0.1 THEN//open
		IF r1.6 THEN//if opened
			r0.1 := 0;
		ELSE
			r0.0 := 0;
			r0.2 := 0;
		END_IF;
	END_IF;

	IF r0.2 THEN
		IF NOT MB.Status.2 THEN
			r0.2 := 0;
		ELSE
			r0.0 := 0;
			r0.1 := 0;
		END_IF;
	END_IF;

	IF MBMOpen_0.ident = 0 THEN
		MBMOpen_0(enable := TRUE, pDevice := pDevice, pMode := ADR('/PHY=RS485 /PA=N /DB=8 /SB=1 /BD=9600'), timeout := 1500);
	ELSE
		IF MBMOpen_0.status = 0 THEN
			CASE step OF
				0:MBMCmd_0(enable := TRUE,ident := MBMOpen_0.ident, mfc := 3, node := 1, offset := 3001, len := 1, data := ADR(MB.Status));
					IF MBMCmd_0.status = 0 THEN
						step := 1;
					END_IF
				1:MBMCmd_0(enable := TRUE,ident := MBMOpen_0.ident, mfc  := 3, node := 1, offset := 3004, len:= 1, data := ADR(MB.Cur_Position));
					IF MBMCmd_0.status = 0 THEN
						Get_Position := MB.Cur_Position;
						step := 2;
					END_IF
				2:IF MB.Commands <> r0 THEN
						MBMCmd_0(enable := TRUE,ident := MBMOpen_0.ident, mfc  := 6, node := 1, offset := 3006, len := 1, data := ADR(r0));
						IF MBMCmd_0.status = 0 THEN
							MB.Commands := r0;
							step := 3;
						END_IF
					ELSE
						step := 3;
					END_IF
				3:IF MB.Set_Position <> Set_Position THEN
						MBMCmd_0(enable := TRUE,ident := MBMOpen_0.ident, mfc  := 6, node := 1, offset := 3007, len := 1, data := ADR(Set_Position));
						IF MBMCmd_0.status = 0 THEN
							MB.Set_Position := Set_Position;
							step := 0;
						END_IF
					ELSE
						step := 0;
					END_IF
				ELSE step := 0;
			END_CASE
		ELSE
			MBMClose_0(enable := TRUE, ident := MBMOpen_0.ident);
			MBMOpen_0(enable := TRUE, pDevice := pDevice, pMode := ADR('/PHY=RS485 /PA=N /DB=8 /SB=1 /BD=9600'), timeout := 1500);
		END_IF
	END_IF

	r1.2 := MB.Status.5; //REMOTE
	r1.3 := MB.Status.4; //LOCAL
	r1.4 := MB.Status.2 AND r0.0; //OPENING
	r1.5 := MB.Status.2 AND r0.1; //CLOSING
	r1.6 := MB.Status.1; //OPENED
	r1.7 := MB.Status.0; //CLOSED
	IF MBMCmd_0.status = 20220 THEN //NOT RESPONSE
		r1.11 := TRUE;
	ELSIF MBMCmd_0.status = 0 THEN
		r1.11 := FALSE;
	END_IF

END_FUNCTION_BLOCK
```

#### LibIP001.fun - Exported functions and function blocks
```iecst
{REDUND_OK} FUNCTION_BLOCK Valve_Biffi (*Biffi valve modbus*) (*$GROUP=User,$CAT=User,$GROUPICON=User.png,$CATICON=User.png*)
	VAR_INPUT
		pDevice : UDINT;
		r0 : UINT;
		Set_Position : UINT;
	END_VAR
	VAR_OUTPUT
		Failures : UINT;
		r1 : UINT;
		Get_Position : UINT;
	END_VAR
	VAR
		MBMOpen_0 : MBMOpen;
		MBMClose_0 : MBMClose;
		MBMCmd_0 : MBMCmd;
		MB : Biffi_Data;
		step : USINT;
	END_VAR
END_FUNCTION_BLOCK

{REDUND_OK} FUNCTION_BLOCK Level_Insol (*Insol Level Sensor Modbus*) (*$GROUP=User,$CAT=User,$GROUPICON=User.png,$CATICON=User.png*)
	VAR_INPUT
		pDevice : UDINT;
	END_VAR
END_FUNCTION_BLOCK

{REDUND_OK} FUNCTION_BLOCK Valve_XCH (*Xenchun valve modbus*) (*$GROUP=User,$CAT=User,$GROUPICON=User.png,$CATICON=User.png*)
	VAR_INPUT
		pDevice : UDINT;
		r0 : UINT;
		Set_Position : UINT;
	END_VAR
	VAR_OUTPUT
		Failures : UINT;
		r1 : UINT;
		Get_Position : UINT;
	END_VAR
	VAR
		MBMOpen_0 : MBMOpen;
		MBMClose_0 : MBMClose;
		MBMCmd_0 : MBMCmd;
		MB : Biffi_Data;
		step : USINT;
		cmd_buf : UINT;
	END_VAR
END_FUNCTION_BLOCK

{REDUND_OK} FUNCTION_BLOCK Valves_XCH (* *) (*$CAT=User,$GROUPICON=User.png,$CATICON=User.png*)
	VAR_INPUT
		pDevice : UDINT;
		r0_2 : UINT;
		r0_1 : UINT;
		Set_Position_2 : UINT;
		Set_Position_1 : UINT;
	END_VAR
	VAR_OUTPUT
		Failures_2 : UINT;
		Failures_1 : UINT;
		r1_2 : UINT;
		r1_1 : UINT;
		Get_Position_2 : UINT;
		Get_Position_1 : UINT;
	END_VAR
	VAR
		MBMOpen_0 : MBMOpen;
		MBMClose_0 : MBMClose;
		MBMCmd_0 : MBMCmd;
		MB_2 : Biffi_Data;
		MB_1 : Biffi_Data;
		step : USINT;
		cmd_buf_2 : UINT;
		cmd_buf_1 : UINT;
	END_VAR
END_FUNCTION_BLOCK

{REDUND_OK} FUNCTION_BLOCK Valves_Biffi
	VAR_INPUT
		pDevice : UDINT;
		r0_1 : UINT;
		r0_2 : UINT;
		Set_Position_1 : UINT;
		Set_Position_2 : UINT;
	END_VAR
	VAR_OUTPUT
		r1_1 : UINT;
		r1_2 : UINT;
		Failures_1 : UINT;
		Failures_2 : UINT;
		Get_Position_1 : UINT;
		Get_Position_2 : UINT;
	END_VAR
	VAR
		MB_1 : Biffi_Data;
		MB_2 : Biffi_Data;
		MBMOpen_0 : MBMOpen;
		MBMClose_0 : MBMClose;
		MBMCmd_0 : MBMCmd;
		step : USINT;
	END_VAR
END_FUNCTION_BLOCK
```

#### Level_Insol.st
```iecst
(* Insol Level Sensor Modbus *)
FUNCTION_BLOCK Level_Insol
END_FUNCTION_BLOCK
```

#### Valve_XCH.st
```iecst
(* Xenchun valve modbus *)
FUNCTION_BLOCK Valve_XCH

	(* Блокировка неактуальных команд *)
	IF r0.0 AND r1.6 THEN
		r0.0 := 0;
	ELSE
		r0.1 := 0;
		r0.2 := 0;
	END_IF;
	IF r0.1 AND r1.7 THEN
		r0.1 := 0;
	ELSE
		r0.0 := 0;
		r0.2 := 0;
	END_IF;
	IF r0.2 AND NOT MB.Status.2 THEN
		r0.2 := 0;
	ELSE
		r0.0 := 0;
		r0.1 := 0;
	END_IF;

	cmd_buf.0 := r0.2;
	cmd_buf.1 := r0.1;
	cmd_buf.10 := r0.0;

	IF MBMOpen_0.ident = 0 THEN
		MBMOpen_0(enable := TRUE, pDevice := pDevice, pMode := ADR('/PHY=RS485 /PA=N /DB=8 /SB=1 /BD=9600'), timeout := 1500);
	END_IF
	IF MBMOpen_0.status = 0 THEN
			CASE step OF
				0:MBMCmd_0(enable := TRUE,ident := MBMOpen_0.ident, mfc := 4, node := 1, offset := 3, len := 1, data := ADR(MB.Status));
					IF MBMCmd_0.status = 0 THEN
						step := 1;
					END_IF
				1:MBMCmd_0(enable := TRUE,ident := MBMOpen_0.ident, mfc  := 4, node := 1, offset := 2, len:= 1, data := ADR(MB.Cur_Position));
					IF MBMCmd_0.status = 0 THEN
						step := 2;
					END_IF
				2:IF MB.Commands <> r0 THEN
						MBMCmd_0(enable := TRUE,ident := MBMOpen_0.ident, mfc  := 6, node := 1, offset := 1, len := 1, data := ADR(cmd_buf));
						IF MBMCmd_0.status = 0 THEN
							MB.Commands := cmd_buf;
							step := 3;
						END_IF
					ELSE
						step := 3;
					END_IF
				3:IF MB.Set_Position <> Set_Position THEN
						MBMCmd_0(enable := TRUE,ident := MBMOpen_0.ident, mfc  := 6, node := 1, offset := 2, len := 1, data := ADR(Set_Position));
						IF MBMCmd_0.status = 0 THEN
							MB.Set_Position := Set_Position;
							step := 0;
						END_IF
					ELSE
						step := 0;
					END_IF
				ELSE step := 0;
			END_CASE
	ELSE
		MBMClose_0(enable := TRUE, ident := MBMOpen_0.ident);
		MBMOpen_0(enable := TRUE, pDevice := pDevice, pMode := ADR('/PHY=RS485 /PA=N /DB=8 /SB=1 /BD=9600'), timeout := 1500);
	END_IF

	r1.2 := MB.Status.1; //REMOTE
	r1.3 := NOT MB.Status.1; //LOCAL
	r1.4 := MB.Status.2; //OPENING
	r1.5 := MB.Status.3; //CLOSING
	r1.6 := MB.Status.5; //OPENED
	r1.7 := MB.Status.4; //CLOSED
	IF MBMCmd_0.status = 20220 THEN //NOT RESPONSE
		r1.11 := TRUE;
	ELSIF MBMCmd_0.status = 0 THEN
		r1.11 := FALSE;
	END_IF

END_FUNCTION_BLOCK
```

#### Valves_XCH.st
```iecst
(* Xenchun valves modbus *)
FUNCTION_BLOCK Valves_XCH

	(* Блокировка неактуальных команд *)
	IF r0_1.0 AND r1_1.6 THEN
		r0_1.0 := 0;
	ELSIF r0_1.0 <> cmd_buf_1.1 THEN
		r0_1.1 := 0;
		r0_1.2 := 0;
	END_IF;
	IF r0_1.1 AND r1_1.7 THEN
		r0_1.1 := 0;
	ELSIF r0_1.1 <> cmd_buf_1.0 THEN
		r0_1.0 := 0;
		r0_1.2 := 0;
	END_IF;
	IF r0_1.2 AND NOT MB_1.Status.2 THEN
		r0_1.2 := 0;
	END_IF;

	cmd_buf_1.0 := r0_1.1;//закрыть
	cmd_buf_1.1 := r0_1.0;//открыть
	IF r0_1.2 THEN 		//stop
		cmd_buf_1.0 := 0;
		cmd_buf_1.1 := 0;
	END_IF

	//Valve 2
	IF r0_2.0 AND r1_2.6 THEN
		r0_2.0 := 0;
	ELSIF r0_2.0 <> cmd_buf_2.1 THEN
		r0_2.1 := 0;
		r0_2.2 := 0;
	END_IF;
	IF r0_2.1 AND r1_2.7 THEN
		r0_2.1 := 0;
	ELSIF r0_2.1 <> cmd_buf_2.0 THEN
		r0_2.0 := 0;
		r0_2.2 := 0;
	END_IF;
	IF r0_2.2 AND NOT MB_2.Status.2 THEN
		r0_2.2 := 0;
	END_IF;

	cmd_buf_2.0 := r0_2.1;//закрыть
	cmd_buf_2.1 := r0_2.0;//открыть
	IF r0_2.2 THEN 		//stop
		cmd_buf_2.0 := 0;
		cmd_buf_2.1 := 0;
	END_IF

	IF MBMOpen_0.ident = 0 THEN
		MBMOpen_0(enable := TRUE, pDevice := pDevice, pMode := ADR('/PHY=RS485 /PA=N /DB=8 /SB=1 /BD=9600'), timeout := 1500);
	END_IF
	IF MBMOpen_0.status = 0 THEN
		CASE step OF
			0:MBMCmd_0(enable := TRUE,ident := MBMOpen_0.ident, mfc := 4, node := 1, offset := 2, len := 1, data := ADR(MB_1.Status));
				IF MBMCmd_0.status <> ERR_FUB_BUSY THEN
					step := 1;
				END_IF
			1:MBMCmd_0(enable := TRUE,ident := MBMOpen_0.ident, mfc  := 4, node := 1, offset := 1, len:= 1, data := ADR(MB_1.Cur_Position));
				IF MBMCmd_0.status <> ERR_FUB_BUSY  THEN
					step := 2;
				END_IF
			2:IF MB_1.Commands <> r0_1 THEN
					MBMCmd_0(enable := TRUE,ident := MBMOpen_0.ident, mfc  := 6, node := 1, offset := 0, len := 1, data := ADR(cmd_buf_1));
					IF MBMCmd_0.status <> ERR_FUB_BUSY  THEN
						MB_1.Commands := cmd_buf_1;
						step := 3;
					END_IF
				ELSE
					step := 3;
				END_IF
			3:IF MB_1.Set_Position <> Set_Position_1 THEN
					Set_Position_1.15 := 0;
					Set_Position_1.14 := 1;
					MBMCmd_0(enable := TRUE,ident := MBMOpen_0.ident, mfc  := 6, node := 1, offset := 1, len := 1, data := ADR(Set_Position_1));
					IF MBMCmd_0.status <> ERR_FUB_BUSY THEN
						MB_1.Set_Position := Set_Position_1;
						step := 4;
					END_IF
				ELSE
					step := 4;
				END_IF

			4: MBMCmd_0(enable := TRUE,ident := MBMOpen_0.ident, mfc := 4, node := 2, offset := 2, len := 1, data := ADR(MB_2.Status));
				IF MBMCmd_0.status <> ERR_FUB_BUSY THEN
					step := 5;
				END_IF
			5:MBMCmd_0(enable := TRUE,ident := MBMOpen_0.ident, mfc  := 4, node := 2, offset := 1, len:= 1, data := ADR(MB_2.Cur_Position));
				IF MBMCmd_0.status <> ERR_FUB_BUSY THEN
					step := 6;
				END_IF
			6:IF MB_2.Commands <> r0_2 THEN
					MBMCmd_0(enable := TRUE,ident := MBMOpen_0.ident, mfc  := 6, node := 2, offset := 0, len := 1, data := ADR(cmd_buf_2));
					IF MBMCmd_0.status <> ERR_FUB_BUSY THEN
						MB_2.Commands := cmd_buf_2;
						step := 7;
					END_IF
				ELSE
					step := 7;
				END_IF
			7:IF MB_2.Set_Position <> Set_Position_2 THEN
					Set_Position_2.15 := 0;
					Set_Position_2.14 := 1;
					MBMCmd_0(enable := TRUE,ident := MBMOpen_0.ident, mfc  := 6, node := 2, offset := 1, len := 1, data := ADR(Set_Position_2));
					IF MBMCmd_0.status <> ERR_FUB_BUSY THEN
						MB_2.Set_Position := Set_Position_2;
						step := 0;
					END_IF
				ELSE
					step := 0;
				END_IF
			ELSE step := 0;
		END_CASE
	ELSE
		MBMClose_0(enable := TRUE, ident := MBMOpen_0.ident);
		MBMOpen_0(enable := TRUE, pDevice := pDevice, pMode := ADR('/PHY=RS485 /PA=N /DB=8 /SB=1 /BD=9600'), timeout := 1500);
	END_IF

	r1_1.2 := MB_1.Status.1; //REMOTE
	r1_1.3 := NOT MB_1.Status.1; //LOCAL
	r1_1.4 := MB_1.Status.2; //OPENING
	r1_1.5 := MB_1.Status.3; //CLOSING
	r1_1.6 := MB_1.Status.5; //OPENED
	r1_1.7 := MB_1.Status.4; //CLOSED
	IF (MBMCmd_0.status = 20220 AND step <4) THEN //NOT RESPONSE
		r1_1.11 := TRUE;
	ELSIF (MBMCmd_0.status = 0 AND step <4 )THEN
		r1_1.11 := FALSE;
	END_IF

	r1_2.2 := MB_2.Status.1; //REMOTE
	r1_2.3 := NOT MB_2.Status.1; //LOCAL
	r1_2.4 := MB_2.Status.2; //OPENING
	r1_2.5 := MB_2.Status.3; //CLOSING
	r1_2.6 := MB_2.Status.5; //OPENED
	r1_2.7 := MB_2.Status.4; //CLOSED
	IF (MBMCmd_0.status = 20220 AND step > 4) THEN //NOT RESPONSE
		r1_2.11 := TRUE;
	ELSIF (MBMCmd_0.status = 0 AND step > 4 )THEN
		r1_2.11 := FALSE;
	END_IF
END_FUNCTION_BLOCK
```

#### Valves_Biffi.st
```iecst
(*  *)
FUNCTION_BLOCK Valves_Biffi

(* Biffi valve modbus *)
(*
бит0-закрыть
бит1-открыть
бит2-стоп
бит4-управление положением
*)
	(* Блокировка неактуальных команд *)
	IF r0_1.0 THEN//close
			IF r1_1.7 THEN// if closed
				r0_1.0 := 0;
			ELSE
				r0_1.1 := 0;
				r0_1.2 := 0;
			END_IF;
		END_IF;

		IF r0_1.1 THEN//open
			IF r1_1.6 THEN//if opened
				r0_1.1 := 0;
			ELSE
				r0_1.0 := 0;
				r0_1.2 := 0;
			END_IF;
		END_IF;

		IF r0_1.2 THEN
			IF NOT MB_1.Status.2 THEN
				r0_1.2 := 0;
			ELSE
				r0_1.0 := 0;
				r0_1.1 := 0;
			END_IF;
	END_IF;

	IF r0_2.0 THEN//close
		IF r1_2.7 THEN// if closed
			r0_2.0 := 0;
		ELSE
			r0_2.1 := 0;
			r0_2.2 := 0;
		END_IF;
	END_IF;

	IF r0_2.1 THEN//open
		IF r1_2.6 THEN//if opened
			r0_2.1 := 0;
		ELSE
			r0_2.0 := 0;
			r0_2.2 := 0;
		END_IF;
	END_IF;

	IF r0_2.2 THEN
		IF NOT MB_2.Status.2 THEN
			r0_2.2 := 0;
		ELSE
			r0_2.0 := 0;
			r0_2.1 := 0;
		END_IF;
	END_IF;

		IF MBMOpen_0.ident = 0 THEN
			MBMOpen_0(enable := TRUE, pDevice := pDevice, pMode := ADR('/PHY=RS485 /PA=N /DB=8 /SB=1 /BD=9600'), timeout := 1500);
		ELSE
			IF MBMOpen_0.status = 0 THEN
				CASE step OF
					//valve 1
					0:MBMCmd_0(enable := TRUE,ident := MBMOpen_0.ident, mfc := 3, node := 1, offset := 3001, len := 1, data := ADR(MB_1.Status));
						IF MBMCmd_0.status = 0 THEN
							step := 1;
						END_IF
					1:MBMCmd_0(enable := TRUE,ident := MBMOpen_0.ident, mfc  := 3, node := 1, offset := 3004, len:= 1, data := ADR(MB_1.Cur_Position));
						IF MBMCmd_0.status = 0 THEN
							Get_Position_1 := MB_1.Cur_Position;
							step := 2;
						END_IF
					2:IF MB_1.Commands <> r0_1 THEN
							MBMCmd_0(enable := TRUE,ident := MBMOpen_0.ident, mfc  := 6, node := 1, offset := 3006, len := 1, data := ADR(r0_1));
							IF MBMCmd_0.status = 0 THEN
								MB_1.Commands := r0_1;
								step := 3;
							END_IF
						ELSE
							step := 3;
						END_IF
					3:IF MB_1.Set_Position <> Set_Position_1 THEN
							MBMCmd_0(enable := TRUE,ident := MBMOpen_0.ident, mfc  := 6, node := 1, offset := 3007, len := 1, data := ADR(Set_Position_1));
							IF MBMCmd_0.status = 0 THEN
								MB_1.Set_Position := Set_Position_1;
								step := 0;
							END_IF
						ELSE
							step :=4;
						END_IF
					//valve 2
					4:MBMCmd_0(enable := TRUE,ident := MBMOpen_0.ident, mfc := 3, node := 2, offset := 3001, len := 1, data := ADR(MB_2.Status));
						IF MBMCmd_0.status = 0 THEN
							step := 5;
						END_IF
					5:MBMCmd_0(enable := TRUE,ident := MBMOpen_0.ident, mfc  := 3, node := 2, offset := 3004, len:= 1, data := ADR(MB_2.Cur_Position));
						IF MBMCmd_0.status = 0 THEN
							Get_Position_2 := MB_2.Cur_Position;
							step := 6;
						END_IF
					6:IF MB_2.Commands <> r0_2 THEN
							MBMCmd_0(enable := TRUE,ident := MBMOpen_0.ident, mfc  := 6, node := 2, offset := 3006, len := 1, data := ADR(r0_2));
							IF MBMCmd_0.status = 0 THEN
								MB_2.Commands := r0_2;
								step := 7;
							END_IF
						ELSE
							step := 7;
						END_IF
					7:IF MB_2.Set_Position <> Set_Position_2 THEN
							MBMCmd_0(enable := TRUE,ident := MBMOpen_0.ident, mfc  := 6, node := 2, offset := 3007, len := 1, data := ADR(Set_Position_2));
							IF MBMCmd_0.status = 0 THEN
								MB_2.Set_Position := Set_Position_2;
								step := 0;
							END_IF
						ELSE
							step :=0;
						END_IF
					ELSE step :=0;
				END_CASE
			ELSE
				MBMClose_0(enable := TRUE, ident := MBMOpen_0.ident);
				MBMOpen_0(enable := TRUE, pDevice := pDevice, pMode := ADR('/PHY=RS485 /PA=N /DB=8 /SB=1 /BD=9600'), timeout := 1500);
			END_IF
		END_IF
		// valve1
		r1_1.2 := MB_1.Status.5; //REMOTE
		r1_1.3 := MB_1.Status.4; //LOCAL
		r1_1.4 := MB_1.Status.2 AND r0_1.0; //OPENING
		r1_1.5 := MB_1.Status.2 AND r0_1.1; //CLOSING
		r1_1.6 := MB_1.Status.1; //OPENED
		r1_1.7 := MB_1.Status.0; //CLOSED
		IF MBMCmd_0.status = 20220 THEN //NOT RESPONSE
			r1_1.11 := TRUE;
		ELSIF MBMCmd_0.status = 0 THEN
			r1_1.11 := FALSE;
		END_IF
	// valve2
		r1_2.2 := MB_2.Status.5; //REMOTE
		r1_2.3 := MB_2.Status.4; //LOCAL
		r1_2.4 := MB_2.Status.2 AND r0_2.0; //OPENING
		r1_2.5 := MB_2.Status.2 AND r0_2.1; //CLOSING
		r1_2.6 := MB_2.Status.1; //OPENED
		r1_2.7 := MB_2.Status.0; //CLOSED
		IF MBMCmd_0.status = 20220 THEN //NOT RESPONSE
			r1_2.11 := TRUE;
		ELSIF MBMCmd_0.status = 0 THEN
			r1_2.11 := FALSE;
		END_IF

END_FUNCTION_BLOCK

END_FUNCTION_BLOCK
```

### Program Logical/DCS2_2 (IEC) - Блок манифольда

#### Variables.var
```iecst
VAR CONSTANT
	def_AI_MC : USINT := 1; (*Количество модулей AI*)
	def_AI_WC : USINT := 8; (*Количество входов в AI*)
	def_AO_MC : USINT := 1; (*Количество модулей AO*)
	def_AO_WC : USINT := 1; (*Количество входов в AO*)
	def_DI_MC : USINT := 1; (*Количество модулей DI*)
	def_DI_WC : USINT := 4; (*Количество входов в DI*)
	def_DO_MC : USINT := 1; (*Количество модулей DO*)
	def_DO_WC : USINT := 6; (*Количество входов в DO*)
END_VAR
VAR
	AI : ARRAY[1..def_AI_MC,1..def_AI_WC] OF FAI;
	AO : ARRAY[1..def_AO_MC,1..def_AO_WC] OF FAO;
	DI : ARRAY[1..def_DI_MC,1..def_DI_WC] OF FDI;
	DO_ : ARRAY[1..def_DO_MC,1..def_DO_WC] OF FDO;
	i : USINT;
	j : USINT;
	PostGAS : FPostGassing;
	PAZ : FAlarm;
	XV01 : Valves_Biffi;
END_VAR
```

#### Main.st
```iecst
PROGRAM _INIT
	AI[1,1].LoScale := 0; 	AI[1,1].HiScale := 1.6;
	AI[1,1].RegCmd := 0;

	AI[1,2].LoScale := -50; 	AI[1,2].HiScale := 150;
	AI[1,2].RegCmd := 0;

	AI[1,3].LoScale := -50; 	AI[1,3].HiScale := 150;
	AI[1,3].RegCmd := 0;

	AI[1,6].LoScale := 0; 	AI[1,6].HiScale := 100;
	AI[1,6].HiLimit := 20; 	AI[1,6].HiHiLimit := 50;
	AI[1,6].RegCmd := 48;

	PAZ.EN := 1;
	PAZ.Delay := 30;
END_PROGRAM

PROGRAM _CYCLIC
	FOR i := 1 TO def_AI_MC DO
		FOR j := 1 TO def_AI_WC DO
			AI[i,j]();
		END_FOR
	END_FOR
	FOR i := 1 TO def_AO_MC DO
		FOR j := 1 TO def_AO_WC DO
			AO[i,j]();
		END_FOR
	END_FOR
	FOR i := 1 TO def_DI_MC DO
		FOR j := 1 TO def_DI_WC DO
			DI[i,j]();
		END_FOR
	END_FOR
	FOR i := 1 TO def_DO_MC DO
		FOR j := 1 TO def_DO_WC DO
			DO_[i,j]();
		END_FOR
	END_FOR
	//Оповещение загазованности
	PostGAS(StatusAI := AI[1,6].RegStatus);
	DO_[1,1].In := PostGAS.HL01;						//Порог1
	DO_[1,2].In := PostGAS.HL02;						//Порог2
	//Отключение питания по Порог2
	PAZ.IN.0 :=  AI[1,6].HiHiAlarm;
	PAZ(Ack := NOT AI[1,6].HiHiAlarm);
	DO_[1,6].In := PAZ.OUT;
	//Задвижки
	XV01(pDevice := ADR('IF6.ST1.IF1'));
END_PROGRAM

PROGRAM _EXIT

END_PROGRAM
```

### Program Logical/DCS4_1 (IEC) - Блок ВС-2

#### Variables.var
```iecst
VAR CONSTANT
	def_AI_MC : USINT := 2; (*Количество модулей AI*)
	def_AI_WC : USINT := 8; (*Количество входов в AI*)
	def_AO_MC : USINT := 1; (*Количество модулей AO*)
	def_AO_WC : USINT := 4; (*Количество входов в AO*)
	def_DI_MC : USINT := 2; (*Количество модулей DI*)
	def_DI_WC : USINT := 16; (*Количество входов в DI*)
	def_DO_MC : USINT := 1; (*Количество модулей DO*)
	def_DO_WC : USINT := 8; (*Количество входов в DO*)
END_VAR
VAR
	AI : ARRAY[1..def_AI_MC,1..def_AI_WC] OF FAI;
	AO : ARRAY[1..def_AO_MC,1..def_AO_WC] OF FAO;
	DI : ARRAY[1..def_DI_MC,1..def_DI_WC] OF FDI;
	DO_ : ARRAY[1..def_DO_MC,1..def_DO_WC] OF FDO;
	i : USINT;
	j : USINT;
	PostGAS : FPostGassing;
	PAZ : FAlarm;
	PCV4_1 : FPIDreg_r;
	PCV4_2 : FPIDreg_r;
	LCV4_1 : FPIDreg_r;
	LCV4_2 : FPIDreg_r;
	UVP_1 : UVP_TCP;
	XV01 : Valve_Biffi;
	LT01 : Level_Insol;
END_VAR
```

#### Main.st
```iecst
PROGRAM _INIT

END_PROGRAM

PROGRAM _CYCLIC
	FOR i := 1 TO def_AI_MC DO
		FOR j := 1 TO def_AI_WC DO
			AI[i,j]();
		END_FOR
	END_FOR
	FOR i := 1 TO def_AO_MC DO
		FOR j := 1 TO def_AO_WC DO
			AO[i,j]();
		END_FOR
	END_FOR
	FOR i := 1 TO def_DI_MC DO
		FOR j := 1 TO def_DI_WC DO
			DI[i,j]();
		END_FOR
	END_FOR
	FOR i := 1 TO def_DO_MC DO
		FOR j := 1 TO def_DO_WC DO
			DO_[i,j]();
		END_FOR
	END_FOR
	//Оповещение загазованности
	PostGAS(StatusAI := AI[1,7].RegStatus);
	DO_[1,5].In := PostGAS.HL01;						//Порог1
	DO_[1,6].In := PostGAS.HL02;						//Порог2
	//Отключение питания по Порог2
	PAZ.IN.0 :=  AI[1,6].HiHiAlarm;
	PAZ(Ack := NOT AI[1,6].HiHiAlarm);
	DO_[1,5].In := PAZ.OUT;

	//Регулятор давления в НГС
	PCV4_1(X := AI[1,1].Value, Y := AI[2,1].Value);
	AO[1,1].Value := PCV4_1.Y_out;
	//Регулятор давления в НГС
	PCV4_2(X := AI[1,1].Value, Y := AI[2,2].Value);
	AO[1,2].Value := PCV4_2.Y_out;
	//Регулятор уровня в НГС
	LCV4_1(X := AI[1,3].Value, Y := AI[2,3].Value);
	AO[1,3].Value := LCV4_1.Y_out;
	//Регулятор уровня в НГС
	LCV4_2(X := AI[1,4].Value, Y := AI[2,4].Value);
	AO[1,4].Value := LCV4_2.Y_out;
	//Задвижки
	XV01(pDevice := ADR('IF6.ST7.IF1'));
	//Обмен с УВП
	UVP_1(pPort := ADR("IF1.ST1"));
	//Уровнемер ИНСОЛ 901
	LT01(pDevice := ADR('IF6.ST8.IF1'));
END_PROGRAM

PROGRAM _EXIT

END_PROGRAM
```

### Program Logical/DCS5_1 (IEC) - Блок С-1

#### Variables.var
```iecst
VAR CONSTANT
	def_AI_MC : USINT := 2; (*Количество модулей AI*)
	def_AI_WC : USINT := 8; (*Количество входов в AI*)
	def_AO_MC : USINT := 1; (*Количество модулей AO*)
	def_AO_WC : USINT := 4; (*Количество входов в AO*)
	def_DI_MC : USINT := 2; (*Количество модулей DI*)
	def_DI_WC : USINT := 16; (*Количество входов в DI*)
	def_DO_MC : USINT := 1; (*Количество модулей DO*)
	def_DO_WC : USINT := 8; (*Количество входов в DO*)
END_VAR
VAR
	AI : ARRAY[1..def_AI_MC,1..def_AI_WC] OF FAI;
	AO : ARRAY[1..def_AO_MC,1..def_AO_WC] OF FAO;
	DI : ARRAY[1..def_DI_MC,1..def_DI_WC] OF FDI;
	DO_ : ARRAY[1..def_DO_MC,1..def_DO_WC] OF FDO;
	i : USINT;
	j : USINT;
	PostGAS : FPostGassing;
	PAZ : FAlarm;
	LT01 : Level_Insol;
	PCV5_1 : FPIDreg_r;
	LCV5_1 : FPIDreg_r;
	LCV5_2 : FPIDreg_r;
	UVP_1 : UVP_TCP;
END_VAR
```

#### Main.st
```iecst
PROGRAM _INIT
	(* Insert code here *)

END_PROGRAM

PROGRAM _CYCLIC
	FOR i := 1 TO def_AI_MC DO
		FOR j := 1 TO def_AI_WC DO
			AI[i,j]();
		END_FOR
	END_FOR
	FOR i := 1 TO def_AO_MC DO
		FOR j := 1 TO def_AO_WC DO
			AO[i,j]();
		END_FOR
	END_FOR
	FOR i := 1 TO def_DI_MC DO
		FOR j := 1 TO def_DI_WC DO
			DI[i,j]();
		END_FOR
	END_FOR
	FOR i := 1 TO def_DO_MC DO
		FOR j := 1 TO def_DO_WC DO
			DO_[i,j]();
		END_FOR
	END_FOR
	//Оповещение загазованности
	PostGAS(StatusAI := AI[1,6].RegStatus);
	DO_[1,1].In := PostGAS.HL01;						//Порог1
	DO_[1,2].In := PostGAS.HL02;						//Порог2
	//Регулятор давления в C-1
	PCV5_1(X := AI[1,1].Value, Y := AI[2,1].Value);
	AO[1,1].Value := PCV5_1.Y_out;
	//Регулятор уровня в C-1
	LCV5_1(X := AI[1,3].Value, Y := AI[2,2].Value);
	AO[1,2].Value := LCV5_1.Y_out;
	//Регулятор уровня в C-1
	LCV5_2(X := AI[1,4].Value, Y := AI[2,3].Value);
	AO[1,3].Value := LCV5_2.Y_out;
	//Отключение питания по Порог2
	PAZ.IN.0 :=  AI[1,6].HiHiAlarm;
	PAZ(Ack := NOT AI[1,6].HiHiAlarm);
	DO_[1,8].In := PAZ.OUT;
	//Обмен с УВП
	UVP_1(pPort := ADR("IF2.ST1"));
	//Уровнемер ИНСОЛ 901
	LT01(pDevice := ADR('IF6.ST8.IF1'));
END_PROGRAM

PROGRAM _EXIT
	(* Insert code here *)

END_PROGRAM
```

### Program Logical/DCS9_1 (IEC) - Блок ПТГ

#### Variables.var
```iecst
VAR CONSTANT
	def_AI_MC : USINT := 1; (*Количество модулей AI*)
	def_AI_WC : USINT := 8; (*Количество входов в AI*)
	def_AO_MC : USINT := 1; (*Количество модулей AO*)
	def_AO_WC : USINT := 1; (*Количество входов в AO*)
	def_DI_MC : USINT := 1; (*Количество модулей DI*)
	def_DI_WC : USINT := 8; (*Количество входов в DI*)
	def_DO_MC : USINT := 1; (*Количество модулей DO*)
	def_DO_WC : USINT := 8; (*Количество входов в DO*)
END_VAR
VAR
	AI : ARRAY[1..def_AI_MC,1..def_AI_WC] OF FAI;
	AO : ARRAY[1..def_AO_MC,1..def_AO_WC] OF FAO;
	DI : ARRAY[1..def_DI_MC,1..def_DI_WC] OF FDI;
	DO_ : ARRAY[1..def_DO_MC,1..def_DO_WC] OF FDO;
	i : USINT;
	j : USINT;
	PAZ : FAlarm;
	PostGAS : FPostGassing;
	XV01 : Valve_Biffi;
END_VAR
```

#### Main.st
```iecst
PROGRAM _INIT
	(* Insert code here *)

END_PROGRAM

PROGRAM _CYCLIC	FOR i := 1 TO def_AI_MC DO
		FOR j := 1 TO def_AI_WC DO
			AI[i,j]();
		END_FOR
	END_FOR
	FOR i := 1 TO def_AO_MC DO
		FOR j := 1 TO def_AO_WC DO
			AO[i,j]();
		END_FOR
	END_FOR
	FOR i := 1 TO def_DI_MC DO
		FOR j := 1 TO def_DI_WC DO
			DI[i,j]();
		END_FOR
	END_FOR
	FOR i := 1 TO def_DO_MC DO
		FOR j := 1 TO def_DO_WC DO
			DO_[i,j]();
		END_FOR
	END_FOR
	//Оповещение загазованности
	PostGAS(StatusAI := AI[1,6].RegStatus);
	DO_[1,1].In := PostGAS.HL01;						//Порог1
	DO_[1,2].In := PostGAS.HL02;						//Порог2
	//Отключение питания по Порог2
	PAZ.IN.0 :=  AI[1,6].HiHiAlarm;
	PAZ(Ack := NOT AI[1,6].HiHiAlarm);
	DO_[1,8].In := PAZ.OUT;
	//Задвижки
	XV01(pDevice := ADR('IF6.ST5.IF1'));
END_PROGRAM

PROGRAM _EXIT
	(* Insert code here *)

END_PROGRAM
```

### Program Logical/DCS13_1 (IEC) - Блок БЕН-1

#### Variables.var
```iecst
VAR CONSTANT
	def_AI_MC : USINT := 1; (*Количество модулей AI*)
	def_AI_WC : USINT := 8; (*Количество входов в AI*)
	def_AO_MC : USINT := 1; (*Количество модулей AO*)
	def_AO_WC : USINT := 1; (*Количество входов в AO*)
	def_DI_MC : USINT := 1; (*Количество модулей DI*)
	def_DI_WC : USINT := 8; (*Количество входов в DI*)
	def_DO_MC : USINT := 1; (*Количество модулей DO*)
	def_DO_WC : USINT := 6; (*Количество входов в DO*)
END_VAR
VAR
	AI : ARRAY[1..def_AI_MC,1..def_AI_WC] OF FAI;
	AO : ARRAY[1..def_AO_MC,1..def_AO_WC] OF FAO;
	DI : ARRAY[1..def_DI_MC,1..def_DI_WC] OF FDI;
	DO_ : ARRAY[1..def_DO_MC,1..def_DO_WC] OF FDO;
	i : USINT;
	j : USINT;
	PAZ : FAlarm;
	PostGAS : FPostGassing;
	XV0102 : Valves_XCH;
END_VAR
```

#### Main.st
```iecst
PROGRAM _INIT
	AI[1,1].LoScale := 0; 	AI[1,1].HiScale := 1.6;
	AI[1,1].RegCmd := 0;

	AI[1,2].LoScale := -50; 	AI[1,2].HiScale := 150;
	AI[1,2].RegCmd := 0;

	AI[1,3].LoScale := 0; 	AI[1,3].HiScale := 200;
	AI[1,3].RegCmd := 0;

	AI[1,4].LoScale := 0; 	AI[1,4].HiScale := 200;
	AI[1,4].RegCmd := 0;

	AI[1,6].LoScale := 0; 	AI[1,6].HiScale := 100;
	AI[1,6].HiLimit := 20; 	AI[1,6].HiHiLimit := 50;
	AI[1,6].RegCmd := 48;

	PAZ.EN := 1;
	PAZ.Delay := 30;

END_PROGRAM

PROGRAM _CYCLIC
	FOR i := 1 TO def_AI_MC DO
		FOR j := 1 TO def_AI_WC DO
			AI[i,j]();
		END_FOR
	END_FOR
	FOR i := 1 TO def_AO_MC DO
		FOR j := 1 TO def_AO_WC DO
			AO[i,j]();
		END_FOR
	END_FOR
	FOR i := 1 TO def_DI_MC DO
		FOR j := 1 TO def_DI_WC DO
			DI[i,j]();
		END_FOR
	END_FOR
	FOR i := 1 TO def_DO_MC DO
		FOR j := 1 TO def_DO_WC DO
			DO_[i,j]();
		END_FOR
	END_FOR
	//Оповещение загазованности
	PostGAS(StatusAI := AI[1,6].RegStatus);
	DO_[1,1].In := PostGAS.HL01;						//Порог1
	DO_[1,2].In := PostGAS.HL02;						//Порог2
	//Отключение питания по Порог2
	PAZ.IN.0 :=  AI[1,6].HiHiAlarm;
	PAZ(Ack := NOT AI[1,6].HiHiAlarm);
	DO_[1,6].In := PAZ.OUT;
	//Задвижки
	XV0102(pDevice := ADR('IF6.ST1.IF1'));
END_PROGRAM

PROGRAM _EXIT
	(* Insert code here *)

END_PROGRAM
```

### Program Logical/DCS15_1 (IEC) - Блок БЕВ-1

#### Variables.var
```iecst
VAR CONSTANT
	def_AI_MC : USINT := 1; (*Количество модулей AI*)
	def_AI_WC : USINT := 8; (*Количество входов в AI*)
	def_AO_MC : USINT := 1; (*Количество модулей AO*)
	def_AO_WC : USINT := 1; (*Количество входов в AO*)
	def_DI_MC : USINT := 1; (*Количество модулей DI*)
	def_DI_WC : USINT := 8; (*Количество входов в DI*)
	def_DO_MC : USINT := 1; (*Количество модулей DO*)
	def_DO_WC : USINT := 6; (*Количество входов в DO*)
END_VAR
VAR
	AI : ARRAY[1..def_AI_MC,1..def_AI_WC] OF FAI;
	AO : ARRAY[1..def_AO_MC,1..def_AO_WC] OF FAO;
	DI : ARRAY[1..def_DI_MC,1..def_DI_WC] OF FDI;
	DO_ : ARRAY[1..def_DO_MC,1..def_DO_WC] OF FDO;
	i : USINT;
	j : USINT;
	PostGAS : FPostGassing;
	PAZ : FAlarm;
	XV0102 : Valves_XCH;
END_VAR
```

#### Main.st
```iecst
PROGRAM _INIT
	(* Insert code here *)

END_PROGRAM

PROGRAM _CYCLIC
	FOR i := 1 TO def_AI_MC DO
		FOR j := 1 TO def_AI_WC DO
			AI[i,j]();
		END_FOR
	END_FOR
	FOR i := 1 TO def_AO_MC DO
		FOR j := 1 TO def_AO_WC DO
			AO[i,j]();
		END_FOR
	END_FOR
	FOR i := 1 TO def_DI_MC DO
		FOR j := 1 TO def_DI_WC DO
			DI[i,j]();
		END_FOR
	END_FOR
	FOR i := 1 TO def_DO_MC DO
		FOR j := 1 TO def_DO_WC DO
			DO_[i,j]();
		END_FOR
	END_FOR
	//Оповещение загазованности
	PostGAS(StatusAI := AI[1,6].RegStatus);
	DO_[1,1].In := PostGAS.HL01;						//Порог1
	DO_[1,2].In := PostGAS.HL02;						//Порог2
	//Отключение питания по Порог2
	PAZ.IN.0 :=  AI[1,6].HiHiAlarm;
	PAZ(Ack := NOT AI[1,6].HiHiAlarm);
	DO_[1,6].In := PAZ.OUT;
	//Задвижки
	XV0102(pDevice := ADR('IF6.ST1.IF1'));

END_PROGRAM

PROGRAM _EXIT
	(* Insert code here *)

END_PROGRAM
```

### Program Logical/DCS18_1 (IEC) - Блок САУ

#### Types.typ
```iecst
TYPE
	ModBusMaster : 	STRUCT
		MBMOpen : MBMOpen;
		MBMCmd : MBMCmd;
		MBMClose : MBMClose;
		step : USINT;
	END_STRUCT;
END_TYPE
```

#### Variables.var
```iecst
VAR CONSTANT
	def_AI_MC : USINT := 1; (*Количество модулей AI*)
	def_AI_WC : USINT := 8; (*Количество входов в AI*)
	def_AO_MC : USINT := 1; (*Количество модулей AO*)
	def_AO_WC : USINT := 4; (*Количество входов в AO*)
	def_DI_MC : USINT := 6; (*Количество модулей DI*)
	def_DI_WC : USINT := 16; (*Количество входов в DI*)
	def_DO_MC : USINT := 3; (*Количество модулей DO*)
	def_DO_WC : USINT := 16; (*Количество входов в DO*)
END_VAR
VAR
	AI : ARRAY[1..def_AI_MC,1..def_AI_WC] OF FAI;
	AO : ARRAY[1..def_AO_MC,1..def_AO_WC] OF FAO;
	DI : ARRAY[1..def_DI_MC,1..def_DI_WC] OF FDI;
	DO_ : ARRAY[1..def_DO_MC,1..def_DO_WC] OF FDO;
	i : USINT;
	j : USINT;
	PostGAS : FPostGassing;
	PAZ : FAlarm;
	KM : ARRAY[1..30] OF FMotor;
	Master : ARRAY[1..7] OF ModBusMaster;
	test : ARRAY[1..20] OF UINT;
END_VAR
```

#### Main.st
```iecst
PROGRAM _INIT

	Master[1].MBMOpen(enable := TRUE, pDevice := ADR('IF6.ST11.IF1'), pMode := ADR('/PHY=RS485 /PA=N /DB=8 /SB=1 /BD=9600'), timeout := 1500);
	Master[2].MBMOpen(enable := TRUE, pDevice := ADR('IF6.ST11.IF1'), pMode := ADR('/PHY=RS485 /PA=N /DB=8 /SB=1 /BD=9600'), timeout := 1500);
	Master[3].MBMOpen(enable := TRUE, pDevice := ADR('IF6.ST11.IF1'), pMode := ADR('/PHY=RS485 /PA=N /DB=8 /SB=1 /BD=9600'), timeout := 1500);
	Master[4].MBMOpen(enable := TRUE, pDevice := ADR('IF6.ST11.IF1'), pMode := ADR('/PHY=RS485 /PA=N /DB=8 /SB=1 /BD=9600'), timeout := 1500);
	Master[5].MBMOpen(enable := TRUE, pDevice := ADR('IF6.ST11.IF1'), pMode := ADR('/PHY=RS485 /PA=N /DB=8 /SB=1 /BD=9600'), timeout := 1500);
	Master[6].MBMOpen(enable := TRUE, pDevice := ADR('IF6.ST11.IF1'), pMode := ADR('/PHY=RS485 /PA=N /DB=8 /SB=1 /BD=9600'), timeout := 1500);
	Master[7].MBMOpen(enable := TRUE, pDevice := ADR('IF6.ST11.IF1'), pMode := ADR('/PHY=RS485 /PA=N /DB=8 /SB=1 /BD=9600'), timeout := 1500);

END_PROGRAM

PROGRAM _CYCLIC
	FOR i := 1 TO def_AI_MC DO
		FOR j := 1 TO def_AI_WC DO
			AI[i,j]();
		END_FOR
	END_FOR
	FOR i := 1 TO def_AO_MC DO
		FOR j := 1 TO def_AO_WC DO
			AO[i,j]();
		END_FOR
	END_FOR
	FOR i := 1 TO def_DI_MC DO
		FOR j := 1 TO def_DI_WC DO
			DI[i,j]();
		END_FOR
	END_FOR
	FOR i := 1 TO def_DO_MC DO
		FOR j := 1 TO def_DO_WC DO
			DO_[i,j]();
		END_FOR
	END_FOR
	//Оповещение загазованности
	PostGAS(StatusAI := AI[1,7].RegStatus);
	DO_[1,5].In := PostGAS.HL01;						//Порог1
	DO_[1,6].In := PostGAS.HL02;						//Порог2
	//Отключение питания по Порог2
	PAZ.IN.0 :=  AI[1,6].HiHiAlarm;
	PAZ(Ack := NOT AI[1,6].HiHiAlarm);
	DO_[1,5].In := PAZ.OUT;
	//QF4
	KM[1](RunDI := DI[1,4].Out);
	DO_[1,1].In := KM[1].StopDO;
	//QF5
	KM[2](RunDI := DI[1,5].Out);
	DO_[1,2].In := KM[2].StopDO;
	//QF6
	KM[3](RunDI := DI[1,6].Out);
	DO_[1,3].In := KM[3].StopDO;
	//QF7
	KM[4](RunDI := DI[1,7].Out);
	DO_[1,4].In := KM[4].StopDO;
	//QF8
	KM[5](RunDI := DI[1,8].Out);
	DO_[1,5].In := KM[5].StopDO;
	//QF9
	KM[6](RunDI := DI[1,9].Out);
	DO_[1,6].In := KM[6].StopDO;
	//QF10
	KM[7](RunDI := DI[1,10].Out);
	DO_[1,7].In := KM[7].StopDO;
	//QF11
	KM[8](RunDI := DI[1,11].Out);
	DO_[1,8].In := KM[8].StopDO;
	//QF12
	KM[9](RunDI := DI[1,12].Out);
	DO_[1,9].In := KM[9].StopDO;
	//QF13
	KM[10](RunDI := DI[1,13].Out);
	DO_[1,10].In := KM[10].StopDO;
	//QF14
	KM[11](RunDI := DI[1,14].Out);
	DO_[1,11].In := KM[11].StopDO;
	//QF15
	KM[12](RunDI := DI[1,15].Out);
	DO_[1,12].In := KM[12].StopDO;
	//QF18
	KM[13](RunDI := DI[2,2].Out);
	DO_[1,15].In := KM[13].StopDO;
	//QF19
	KM[14](RunDI := DI[2,3].Out);
	DO_[1,16].In := KM[14].StopDO;
	//QF31
	KM[15](RunDI := DI[2,9].Out);
	DO_[2,1].In := KM[15].StopDO;
	//QF32
	KM[16](RunDI := DI[2,10].Out);
	DO_[2,2].In := KM[16].StopDO;
	//QF36
	KM[17](RunDI := DI[2,11].Out);
	DO_[2,3].In := KM[17].StopDO;
	//QF37
	KM[18](RunDI := DI[2,12].Out);
	DO_[2,4].In := KM[18].StopDO;
	//QF38
	KM[19](RunDI := DI[2,13].Out);
	DO_[2,5].In := KM[19].StopDO;
	//QF39
	KM[20](RunDI := DI[2,14].Out);
	DO_[2,6].In := KM[20].StopDO;
	//QF40
	KM[21](RunDI := DI[2,15].Out);
	DO_[2,7].In := KM[21].StopDO;
	//QF41
	KM[22](RunDI := DI[2,16].Out);
	DO_[2,8].In := KM[22].StopDO;
	//QF42
	KM[23](RunDI := DI[3,1].Out);
	DO_[2,9].In := KM[23].StopDO;
	//QF43
	KM[23](RunDI := DI[3,2].Out);
	DO_[2,10].In := KM[23].StopDO;
	//QF44
	KM[24](RunDI := DI[3,3].Out);
	DO_[2,11].In := KM[24].StopDO;
	//QF46
	KM[25](RunDI := DI[3,4].Out);
	DO_[2,12].In := KM[25].StopDO;
	//QF47
	KM[26](RunDI := DI[3,5].Out);
	DO_[2,13].In := KM[26].StopDO;
	//QF23
	KM[27](RunDI := DI[3,9].Out);
	DO_[2,15].In := KM[27].StopDO;
	//QF24
	KM[28](RunDI := 0);
	DO_[2,16].In := KM[28].StopDO;
	//ШИБП
	KM[29](RunDI := DI[3,5].Out);
	DO_[2,13].In := KM[29].StopDO;

	//test обмен с ГФУ и БРГ
	IF Master[1].MBMOpen.status = 0 AND Master[1].MBMOpen.ident <> 0 THEN
		CASE Master[1].step OF
			0:
				Master[1].MBMCmd(enable := TRUE,ident := Master[1].MBMOpen.ident, mfc := 3, node := 1, offset := 1, len := 2, data := ADR(test));
				IF Master[1].MBMCmd.status <> ERR_FUB_BUSY THEN
					Master[1].step := 1;
				END_IF
			ELSE
				Master[1].step := 0;
		END_CASE
	END_IF

	//test обмен с БДР
	IF Master[2].MBMOpen.status = 0 AND Master[2].MBMOpen.ident <> 0 THEN
		CASE Master[2].step OF
			0:
				Master[2].MBMCmd(enable := TRUE,ident := Master[2].MBMOpen.ident, mfc := 3, node := 1, offset := 1, len := 2, data := ADR(test));
				IF Master[2].MBMCmd.status <> ERR_FUB_BUSY THEN
					Master[2].step := 1;
				END_IF
			ELSE
				Master[2].step := 0;
		END_CASE
	END_IF

	//test обмен с П-1/1
	IF Master[3].MBMOpen.status = 0 AND Master[3].MBMOpen.ident <> 0 THEN
		CASE Master[3].step OF
			0:
				Master[3].MBMCmd(enable := TRUE,ident := Master[3].MBMOpen.ident, mfc := 3, node := 1, offset := 1, len := 2, data := ADR(test));
				IF Master[3].MBMCmd.status <> ERR_FUB_BUSY THEN
					Master[3].step := 1;
				END_IF
			ELSE
				Master[3].step := 0;
		END_CASE
	END_IF

	//test обмен с ДЭС
	IF Master[4].MBMOpen.status = 0 AND Master[4].MBMOpen.ident <> 0 THEN
		CASE Master[4].step OF
			0:
				Master[4].MBMCmd(enable := TRUE,ident := Master[4].MBMOpen.ident, mfc := 3, node := 1, offset := 1, len := 2, data := ADR(test));
				IF Master[4].MBMCmd.status <> ERR_FUB_BUSY THEN
					Master[4].step := 1;
				END_IF
			ELSE
				Master[4].step := 0;
		END_CASE
	END_IF

	//test обмен с ГПЭС
	IF Master[5].MBMOpen.status = 0 AND Master[5].MBMOpen.ident <> 0 THEN
		CASE Master[5].step OF
			0:
				Master[5].MBMCmd(enable := TRUE,ident := Master[5].MBMOpen.ident, mfc := 3, node := 1, offset := 1, len := 2, data := ADR(test));
				IF Master[5].MBMCmd.status <> ERR_FUB_BUSY THEN
					Master[5].step := 1;
				END_IF
			ELSE
				Master[5].step := 0;
		END_CASE
	END_IF

	//test обмен с ШНКУ
	IF Master[6].MBMOpen.status = 0 AND Master[6].MBMOpen.ident <> 0 THEN
		CASE Master[6].step OF
			0:
				Master[6].MBMCmd(enable := TRUE,ident := Master[6].MBMOpen.ident, mfc := 3, node := 1, offset := 1, len := 2, data := ADR(test));
				IF Master[6].MBMCmd.status <> ERR_FUB_BUSY THEN
					Master[6].step := 1;
				END_IF
			ELSE
				Master[6].step := 0;
		END_CASE
	END_IF

	//test обмен с ШУЭ
	IF Master[7].MBMOpen.status = 0 AND Master[7].MBMOpen.ident <> 0 THEN
		CASE Master[7].step OF
			0:
				Master[7].MBMCmd(enable := TRUE,ident := Master[7].MBMOpen.ident, mfc := 3, node := 1, offset := 1, len := 2, data := ADR(test));
				IF Master[7].MBMCmd.status <> ERR_FUB_BUSY THEN
					Master[7].step := 1;
				END_IF
			ELSE
				Master[7].step := 0;
		END_CASE
	END_IF

END_PROGRAM

PROGRAM _EXIT

END_PROGRAM
```

### Program Logical/DCS31_1 (IEC) - Блок Е-1/1

#### Variables.var
```iecst
VAR CONSTANT
	def_AI_MC : USINT := 1; (*Количество модулей AI*)
	def_AI_WC : USINT := 4; (*Количество входов в AI*)
	def_AO_MC : USINT := 1; (*Количество модулей AO*)
	def_AO_WC : USINT := 1; (*Количество входов в AO*)
	def_DI_MC : USINT := 1; (*Количество модулей DI*)
	def_DI_WC : USINT := 6; (*Количество входов в DI*)
	def_DO_MC : USINT := 1; (*Количество модулей DO*)
	def_DO_WC : USINT := 4; (*Количество входов в DO*)
END_VAR
VAR
	AI : ARRAY[1..def_AI_MC,1..def_AI_WC] OF FAI;
	AO : ARRAY[1..def_AO_MC,1..def_AO_WC] OF FAO;
	DI : ARRAY[1..def_DI_MC,1..def_DI_WC] OF FDI;
	DO_ : ARRAY[1..def_DO_MC,1..def_DO_WC] OF FDO;
	i : USINT;
	j : USINT;
	PostGAS : FPostGassing;
	PAZ : FAlarm;
	XV01 : Valves_XCH;
END_VAR
```

#### Main.st
```iecst
PROGRAM _INIT

END_PROGRAM

PROGRAM _CYCLIC
	FOR i := 1 TO def_AI_MC DO
		FOR j := 1 TO def_AI_WC DO
			AI[i,j]();
		END_FOR
	END_FOR
	FOR i := 1 TO def_AO_MC DO
		FOR j := 1 TO def_AO_WC DO
			AO[i,j]();
		END_FOR
	END_FOR
	FOR i := 1 TO def_DI_MC DO
		FOR j := 1 TO def_DI_WC DO
			DI[i,j]();
		END_FOR
	END_FOR
	FOR i := 1 TO def_DO_MC DO
		FOR j := 1 TO def_DO_WC DO
			DO_[i,j]();
		END_FOR
	END_FOR
	//Оповещение загазованности
	PostGAS(StatusAI := AI[1,4].RegStatus);
	DO_[1,1].In := PostGAS.HL01;						//Порог1
	DO_[1,2].In := PostGAS.HL02;						//Порог2
	//Отключение питания по Порог2
	PAZ.IN.0 :=  AI[1,4].HiHiAlarm;
	PAZ(Ack := NOT AI[1,4].HiHiAlarm);
	DO_[1,4].In := PAZ.OUT;
	//Задвижки
	XV01(pDevice := ADR('IF6.ST1.IF1'));
END_PROGRAM

PROGRAM _EXIT
	(* Insert code here *)

END_PROGRAM
```

### Program Logical/DCS31_2 (IEC) - Блок Е-1/2

#### Variables.var
```iecst
VAR CONSTANT
	def_AI_MC : USINT := 1; (*Количество модулей AI*)
	def_AI_WC : USINT := 4; (*Количество входов в AI*)
	def_AO_MC : USINT := 1; (*Количество модулей AO*)
	def_AO_WC : USINT := 1; (*Количество входов в AO*)
	def_DI_MC : USINT := 1; (*Количество модулей DI*)
	def_DI_WC : USINT := 6; (*Количество входов в DI*)
	def_DO_MC : USINT := 1; (*Количество модулей DO*)
	def_DO_WC : USINT := 4; (*Количество входов в DO*)
END_VAR
VAR
	AI : ARRAY[1..def_AI_MC,1..def_AI_WC] OF FAI;
	AO : ARRAY[1..def_AO_MC,1..def_AO_WC] OF FAO;
	DI : ARRAY[1..def_DI_MC,1..def_DI_WC] OF FDI;
	DO_ : ARRAY[1..def_DO_MC,1..def_DO_WC] OF FDO;
	i : USINT;
	j : USINT;
	PostGAS : FPostGassing;
	PAZ : FAlarm;
	XV01_02 : Valves_XCH;
END_VAR
```

#### Main.st
```iecst
PROGRAM _INIT
	(* Insert code here *)

END_PROGRAM

PROGRAM _CYCLIC
	FOR i := 1 TO def_AI_MC DO
		FOR j := 1 TO def_AI_WC DO
			AI[i,j]();
		END_FOR
	END_FOR
	FOR i := 1 TO def_AO_MC DO
		FOR j := 1 TO def_AO_WC DO
			AO[i,j]();
		END_FOR
	END_FOR
	FOR i := 1 TO def_DI_MC DO
		FOR j := 1 TO def_DI_WC DO
			DI[i,j]();
		END_FOR
	END_FOR
	FOR i := 1 TO def_DO_MC DO
		FOR j := 1 TO def_DO_WC DO
			DO_[i,j]();
		END_FOR
	END_FOR
	//Оповещение загазованности
	PostGAS(StatusAI := AI[1,4].RegStatus);
	DO_[1,1].In := PostGAS.HL01;						//Порог1
	DO_[1,2].In := PostGAS.HL02;						//Порог2
	//Отключение питания по Порог2
	PAZ.IN.0 :=  AI[1,4].HiHiAlarm;
	PAZ(Ack := NOT AI[1,4].HiHiAlarm);
	DO_[1,4].In := PAZ.OUT;
	//Задвижки
	XV01_02(pDevice := ADR('IF6.ST1.IF1'));

END_PROGRAM

PROGRAM _EXIT
	(* Insert code here *)

END_PROGRAM
```

### Program Logical/DCS31_3 (IEC) - Блок Е-1/3

#### Main.st
```iecst
PROGRAM _INIT
	(* Insert code here *)

END_PROGRAM

PROGRAM _CYCLIC
	FOR i := 1 TO def_AI_MC DO
		FOR j := 1 TO def_AI_WC DO
			AI[i,j]();
		END_FOR
	END_FOR
	FOR i := 1 TO def_AO_MC DO
		FOR j := 1 TO def_AO_WC DO
			AO[i,j]();
		END_FOR
	END_FOR
	FOR i := 1 TO def_DI_MC DO
		FOR j := 1 TO def_DI_WC DO
			DI[i,j]();
		END_FOR
	END_FOR
	FOR i := 1 TO def_DO_MC DO
		FOR j := 1 TO def_DO_WC DO
			DO_[i,j]();
		END_FOR
	END_FOR
	//Оповещение загазованности
	PostGAS(StatusAI := AI[1,4].RegStatus);
	DO_[1,1].In := PostGAS.HL01;						//Порог1
	DO_[1,2].In := PostGAS.HL02;						//Порог2
	//Отключение питания по Порог2
	PAZ.IN.0 :=  AI[1,4].HiHiAlarm;
	PAZ(Ack := NOT AI[1,4].HiHiAlarm);
	DO_[1,4].In := PAZ.OUT;
	//Задвижки
	XV01_02(pDevice := ADR('IF6.ST1.IF1'));
END_PROGRAM

PROGRAM _EXIT
	(* Insert code here *)

END_PROGRAM
```

### Program Logical/DCS31_4 (IEC) - Блок Е-1/4

#### Variables.var
```iecst
VAR CONSTANT
	def_AI_MC : USINT := 1; (*Количество модулей AI*)
	def_AI_WC : USINT := 4; (*Количество входов в AI*)
	def_AO_MC : USINT := 1; (*Количество модулей AO*)
	def_AO_WC : USINT := 1; (*Количество входов в AO*)
	def_DI_MC : USINT := 1; (*Количество модулей DI*)
	def_DI_WC : USINT := 6; (*Количество входов в DI*)
	def_DO_MC : USINT := 1; (*Количество модулей DO*)
	def_DO_WC : USINT := 4; (*Количество входов в DO*)
END_VAR
VAR
	AI : ARRAY[1..def_AI_MC,1..def_AI_WC] OF FAI;
	AO : ARRAY[1..def_AO_MC,1..def_AO_WC] OF FAO;
	DI : ARRAY[1..def_DI_MC,1..def_DI_WC] OF FDI;
	DO_ : ARRAY[1..def_DO_MC,1..def_DO_WC] OF FDO;
	i : USINT;
	j : USINT;
	PostGAS : FPostGassing;
	PAZ : FAlarm;
	XV01_02 : Valves_XCH;
	XV02 : Valve_XCH;
END_VAR
```

### Program Logical/DCS34_1 (IEC) - Блок СИКГ-2

#### Variables.var
```iecst
VAR CONSTANT
	def_AI_MC : USINT := 1; (*Количество модулей AI*)
	def_AI_WC : USINT := 8; (*Количество входов в AI*)
	def_AO_MC : USINT := 1; (*Количество модулей AO*)
	def_AO_WC : USINT := 2; (*Количество входов в AO*)
	def_DI_MC : USINT := 1; (*Количество модулей DI*)
	def_DI_WC : USINT := 8; (*Количество входов в DI*)
	def_DO_MC : USINT := 1; (*Количество модулей DO*)
	def_DO_WC : USINT := 6; (*Количество входов в DO*)
END_VAR
VAR
	AI : ARRAY[1..def_AI_MC,1..def_AI_WC] OF FAI;
	AO : ARRAY[1..def_AO_MC,1..def_AO_WC] OF FAO;
	DI : ARRAY[1..def_DI_MC,1..def_DI_WC] OF FDI;
	DO_ : ARRAY[1..def_DO_MC,1..def_DO_WC] OF FDO;
	i : USINT;
	j : USINT;
	PostGAS : FPostGassing;
	PAZ : FAlarm;
	PCV34_1 : FPIDreg_r;
END_VAR
```

#### Main.st
```iecst
PROGRAM _INIT

END_PROGRAM

PROGRAM _CYCLIC
	FOR i := 1 TO def_AI_MC DO
		FOR j := 1 TO def_AI_WC DO
			AI[i,j]();
		END_FOR
	END_FOR
	FOR i := 1 TO def_AO_MC DO
		FOR j := 1 TO def_AO_WC DO
			AO[i,j]();
		END_FOR
	END_FOR
	FOR i := 1 TO def_DI_MC DO
		FOR j := 1 TO def_DI_WC DO
			DI[i,j]();
		END_FOR
	END_FOR
	FOR i := 1 TO def_DO_MC DO
		FOR j := 1 TO def_DO_WC DO
			DO_[i,j]();
		END_FOR
	END_FOR
	//Оповещение загазованности
	PostGAS(StatusAI := AI[1,6].RegStatus);
	DO_[1,1].In := PostGAS.HL01;						//Порог1
	DO_[1,2].In := PostGAS.HL02;						//Порог2
	//Отключение питания по Порог2
	PAZ.IN.0 :=  AI[1,6].HiHiAlarm;
	PAZ(Ack := NOT AI[1,6].HiHiAlarm);
	DO_[1,6].In := PAZ.OUT;

	//Регулятор давления в НГС
	PCV34_1(X := AI[1,1].Value, Y := AI[1,6].Value);
	AO[1,1].Value := PCV34_1.Y_out;

END_PROGRAM

PROGRAM _EXIT

END_PROGRAM
```

### Program Logical/DCS35_1 (IEC) - Блок СИКГ-3/СИКГ-4

#### Variables.var
```iecst
VAR CONSTANT
	def_AI_MC : USINT := 1; (*Количество модулей AI*)
	def_AI_WC : USINT := 4; (*Количество входов в AI*)
	def_AO_MC : USINT := 1; (*Количество модулей AO*)
	def_AO_WC : USINT := 1; (*Количество входов в AO*)
	def_DI_MC : USINT := 1; (*Количество модулей DI*)
	def_DI_WC : USINT := 6; (*Количество входов в DI*)
	def_DO_MC : USINT := 1; (*Количество модулей DO*)
	def_DO_WC : USINT := 6; (*Количество входов в DO*)
END_VAR
VAR
	AI : ARRAY[1..def_AI_MC,1..def_AI_WC] OF FAI;
	AO : ARRAY[1..def_AO_MC,1..def_AO_WC] OF FAO;
	DI : ARRAY[1..def_DI_MC,1..def_DI_WC] OF FDI;
	DO_ : ARRAY[1..def_DO_MC,1..def_DO_WC] OF FDO;
	i : USINT;
	j : USINT;
	PostGAS : FPostGassing;
	PAZ : FAlarm;
END_VAR
```

#### Main.st
```iecst
PROGRAM _INIT
	(* Insert code here *)

END_PROGRAM

PROGRAM _CYCLIC
	FOR i := 1 TO def_AI_MC DO
		FOR j := 1 TO def_AI_WC DO
			AI[i,j]();
		END_FOR
	END_FOR
	FOR i := 1 TO def_AO_MC DO
		FOR j := 1 TO def_AO_WC DO
			AO[i,j]();
		END_FOR
	END_FOR
	FOR i := 1 TO def_DI_MC DO
		FOR j := 1 TO def_DI_WC DO
			DI[i,j]();
		END_FOR
	END_FOR
	FOR i := 1 TO def_DO_MC DO
		FOR j := 1 TO def_DO_WC DO
			DO_[i,j]();
		END_FOR
	END_FOR
	//Оповещение загазованности
	PostGAS(StatusAI := AI[1,4].RegStatus);
	DO_[1,1].In := PostGAS.HL01;						//Порог1
	DO_[1,2].In := PostGAS.HL02;						//Порог2
	//Отключение питания по Порог2
	PAZ.IN.0 :=  AI[1,4].HiHiAlarm;
	PAZ(Ack := NOT AI[1,4].HiHiAlarm);
	DO_[1,6].In := PAZ.OUT;

END_PROGRAM

PROGRAM _EXIT
	(* Insert code here *)

END_PROGRAM
```

### Program Logical/DCS36_1 (IEC) - Блок ГФУ

#### Variables.var
```iecst
VAR CONSTANT
	def_AI_MC : USINT := 1; (*Количество модулей AI*)
	def_AI_WC : USINT := 8; (*Количество входов в AI*)
	def_AO_MC : USINT := 1; (*Количество модулей AO*)
	def_AO_WC : USINT := 1; (*Количество входов в AO*)
	def_DI_MC : USINT := 1; (*Количество модулей DI*)
	def_DI_WC : USINT := 8; (*Количество входов в DI*)
	def_DO_MC : USINT := 1; (*Количество модулей DO*)
	def_DO_WC : USINT := 12; (*Количество входов в DO*)
END_VAR
VAR
	AI : ARRAY[1..def_AI_MC,1..def_AI_WC] OF FAI;
	AO : ARRAY[1..def_AO_MC,1..def_AO_WC] OF FAO;
	DI : ARRAY[1..def_DI_MC,1..def_DI_WC] OF FDI;
	DO_ : ARRAY[1..def_DO_MC,1..def_DO_WC] OF FDO;
	i : USINT;
	j : USINT;
	PostGAS : FPostGassing;
	Torche_1 : FTorch;
	Torche_2_3 : FTorch;
	Torche_4_5 : FTorch;
	P_GAS_LOW : FAlarm;
END_VAR
```

#### Main.st
```iecst
PROGRAM _INIT
	(* Insert code here *)

END_PROGRAM

PROGRAM _CYCLIC
	FOR i := 1 TO def_AI_MC DO
		FOR j := 1 TO def_AI_WC DO
			AI[i,j]();
		END_FOR
	END_FOR
	FOR i := 1 TO def_AO_MC DO
		FOR j := 1 TO def_AO_WC DO
			AO[i,j]();
		END_FOR
	END_FOR
	FOR i := 1 TO def_DI_MC DO
		FOR j := 1 TO def_DI_WC DO
			DI[i,j]();
		END_FOR
	END_FOR
	FOR i := 1 TO def_DO_MC DO
		FOR j := 1 TO def_DO_WC DO
			DO_[i,j]();
		END_FOR
	END_FOR
	//Оповещение загазованности
	PostGAS(StatusAI := AI[1,6].RegStatus);
	DO_[1,5].In := PostGAS.HL01;						//Порог1
	DO_[1,6].In := PostGAS.HL02;						//Порог2
	//Факел 1
	Torche_1(Di_Fire := AI[1,1].HiHiAlarm, Di_P_gas_low := P_GAS_LOW.OUT, Start :=  DI[1,5].Out,  Stop :=  DI[1,6].Out, Mode_Manual := DI[1,4].Out);
	DO_[1,1].In := Torche_1.Do_Lamp_FireON;
	DO_[1,2].In := Torche_1.Do_Spark;
	//Факел 2 3
	Torche_2_3(Di_Fire := AI[1,2].HiHiAlarm OR AI[1,3].HiHiAlarm, Di_P_gas_low := P_GAS_LOW.OUT, Start :=  DI[1,5].Out,  Stop :=  DI[1,6].Out, Mode_Manual := DI[1,4].Out);
	DO_[1,3].In := Torche_2_3.Do_Lamp_FireON AND AI[1,2].HiHiAlarm;
	DO_[1,4].In := Torche_2_3.Do_Lamp_FireON AND AI[1,3].HiHiAlarm;
	DO_[1,5].In := Torche_2_3.Do_Spark;
	//Факел 4 5
	Torche_4_5(Di_Fire := AI[1,4].HiHiAlarm OR AI[1,5].HiHiAlarm, Di_P_gas_low := P_GAS_LOW.OUT, Start :=  DI[1,5].Out,  Stop :=  DI[1,6].Out, Mode_Manual := DI[1,4].Out);
	DO_[1,6].In := Torche_4_5.Do_Lamp_FireON AND AI[1,4].HiHiAlarm;
	DO_[1,7].In := Torche_4_5.Do_Lamp_FireON AND AI[1,5].HiHiAlarm;

	//Управляем клапаном по трем факелам
	DO_[1,11].In := Torche_1.Do_Valve OR Torche_2_3.Do_Valve OR Torche_4_5.Do_Valve;

END_PROGRAM

PROGRAM _EXIT
	(* Insert code here *)

END_PROGRAM
```

### Program Logical/DCS37_1 (IEC) - Блок СИКВ-1

#### Variables.var
```iecst
VAR CONSTANT
	def_AI_MC : USINT := 1; (*Количество модулей AI*)
	def_AI_WC : USINT := 4; (*Количество входов в AI*)
	def_AO_MC : USINT := 1; (*Количество модулей AO*)
	def_AO_WC : USINT := 1; (*Количество входов в AO*)
	def_DI_MC : USINT := 1; (*Количество модулей DI*)
	def_DI_WC : USINT := 4; (*Количество входов в DI*)
	def_DO_MC : USINT := 1; (*Количество модулей DO*)
	def_DO_WC : USINT := 6; (*Количество входов в DO*)
END_VAR
VAR
	AI : ARRAY[1..def_AI_MC,1..def_AI_WC] OF FAI;
	AO : ARRAY[1..def_AO_MC,1..def_AO_WC] OF FAO;
	DI : ARRAY[1..def_DI_MC,1..def_DI_WC] OF FDI;
	DO_ : ARRAY[1..def_DO_MC,1..def_DO_WC] OF FDO;
	i : USINT;
	j : USINT;
	PostGAS : FPostGassing;
	PAZ : FAlarm;
END_VAR
```

#### Main.st
```iecst
PROGRAM _INIT
	(* Insert code here *)

END_PROGRAM

PROGRAM _CYCLIC
	FOR i := 1 TO def_AI_MC DO
		FOR j := 1 TO def_AI_WC DO
			AI[i,j]();
		END_FOR
	END_FOR
	FOR i := 1 TO def_AO_MC DO
		FOR j := 1 TO def_AO_WC DO
			AO[i,j]();
		END_FOR
	END_FOR
	FOR i := 1 TO def_DI_MC DO
		FOR j := 1 TO def_DI_WC DO
			DI[i,j]();
		END_FOR
	END_FOR
	FOR i := 1 TO def_DO_MC DO
		FOR j := 1 TO def_DO_WC DO
			DO_[i,j]();
		END_FOR
	END_FOR
	//Оповещение загазованности
	PostGAS(StatusAI := AI[1,4].RegStatus);
	DO_[1,1].In := PostGAS.HL01;						//Порог1
	DO_[1,2].In := PostGAS.HL02;						//Порог2
	//Отключение питания по Порог2
	PAZ.IN.0 :=  AI[1,4].HiHiAlarm;
	PAZ(Ack := NOT AI[1,4].HiHiAlarm);
	DO_[1,6].In := PAZ.OUT;

END_PROGRAM

PROGRAM _EXIT
	(* Insert code here *)

END_PROGRAM
```

### Program Logical/DCS39_1 (IEC) - Блок СИКГ-1/СИКГ-5

#### Variables.var
```iecst
VAR CONSTANT
	def_AI_MC : USINT := 1; (*Количество модулей AI*)
	def_AI_WC : USINT := 8; (*Количество входов в AI*)
	def_AO_MC : USINT := 1; (*Количество модулей AO*)
	def_AO_WC : USINT := 2; (*Количество входов в AO*)
	def_DI_MC : USINT := 1; (*Количество модулей DI*)
	def_DI_WC : USINT := 8; (*Количество входов в DI*)
	def_DO_MC : USINT := 1; (*Количество модулей DO*)
	def_DO_WC : USINT := 6; (*Количество входов в DO*)
END_VAR
VAR
	AI : ARRAY[1..def_AI_MC,1..def_AI_WC] OF FAI;
	AO : ARRAY[1..def_AO_MC,1..def_AO_WC] OF FAO;
	DI : ARRAY[1..def_DI_MC,1..def_DI_WC] OF FDI;
	DO_ : ARRAY[1..def_DO_MC,1..def_DO_WC] OF FDO;
	i : USINT;
	j : USINT;
	PostGAS : FPostGassing;
	PAZ : FAlarm;
	PCV39_1 : FPIDreg_r;
	UVP_1 : UVP_TCP;
END_VAR
```

#### Main.st
```iecst
PROGRAM _INIT

END_PROGRAM

PROGRAM _CYCLIC
	FOR i := 1 TO def_AI_MC DO
		FOR j := 1 TO def_AI_WC DO
			AI[i,j]();
		END_FOR
	END_FOR
	FOR i := 1 TO def_AO_MC DO
		FOR j := 1 TO def_AO_WC DO
			AO[i,j]();
		END_FOR
	END_FOR
	FOR i := 1 TO def_DI_MC DO
		FOR j := 1 TO def_DI_WC DO
			DI[i,j]();
		END_FOR
	END_FOR
	FOR i := 1 TO def_DO_MC DO
		FOR j := 1 TO def_DO_WC DO
			DO_[i,j]();
		END_FOR
	END_FOR
	//Оповещение загазованности
	PostGAS(StatusAI := AI[1,7].RegStatus);
	DO_[1,5].In := PostGAS.HL01;						//Порог1
	DO_[1,6].In := PostGAS.HL02;						//Порог2
	//Отключение питания по Порог2
	PAZ.IN.0 :=  AI[1,6].HiHiAlarm;
	PAZ(Ack := NOT AI[1,6].HiHiAlarm);
	DO_[1,5].In := PAZ.OUT;

	//Регулятор давления
	PCV39_1(X := AI[1,1].Value, Y := AI[1,2].Value);
	AO[1,1].Value := PCV39_1.Y_out;

END_PROGRAM

PROGRAM _EXIT

END_PROGRAM
```

### Program Logical/DCS40_1 (IEC) - Блок СИКГ-6

#### Variables.var
```iecst
VAR CONSTANT
	def_AI_MC : USINT := 1; (*Количество модулей AI*)
	def_AI_WC : USINT := 8; (*Количество входов в AI*)
	def_AO_MC : USINT := 1; (*Количество модулей AO*)
	def_AO_WC : USINT := 2; (*Количество входов в AO*)
	def_DI_MC : USINT := 1; (*Количество модулей DI*)
	def_DI_WC : USINT := 8; (*Количество входов в DI*)
	def_DO_MC : USINT := 1; (*Количество модулей DO*)
	def_DO_WC : USINT := 6; (*Количество входов в DO*)
END_VAR
VAR
	AI : ARRAY[1..def_AI_MC,1..def_AI_WC] OF FAI;
	AO : ARRAY[1..def_AO_MC,1..def_AO_WC] OF FAO;
	DI : ARRAY[1..def_DI_MC,1..def_DI_WC] OF FDI;
	DO_ : ARRAY[1..def_DO_MC,1..def_DO_WC] OF FDO;
	i : USINT;
	j : USINT;
	PostGAS : FPostGassing;
	PAZ : FAlarm;
	PCV40_1 : FPIDreg_r;
	UVP_1 : UVP_TCP;
END_VAR
```

#### Main.st
```iecst
PROGRAM _INIT

END_PROGRAM

PROGRAM _CYCLIC
	FOR i := 1 TO def_AI_MC DO
		FOR j := 1 TO def_AI_WC DO
			AI[i,j]();
		END_FOR
	END_FOR
	FOR i := 1 TO def_AO_MC DO
		FOR j := 1 TO def_AO_WC DO
			AO[i,j]();
		END_FOR
	END_FOR
	FOR i := 1 TO def_DI_MC DO
		FOR j := 1 TO def_DI_WC DO
			DI[i,j]();
		END_FOR
	END_FOR
	FOR i := 1 TO def_DO_MC DO
		FOR j := 1 TO def_DO_WC DO
			DO_[i,j]();
		END_FOR
	END_FOR
	//Оповещение загазованности
	PostGAS(StatusAI := AI[1,6].RegStatus);
	DO_[1,5].In := PostGAS.HL01;						//Порог1
	DO_[1,6].In := PostGAS.HL02;						//Порог2
	//Отключение питания по Порог2
	PAZ.IN.0 :=  AI[1,6].HiHiAlarm;
	PAZ(Ack := NOT AI[1,6].HiHiAlarm);
	DO_[1,6].In := PAZ.OUT;

	//Регулятор давления в НГС
	PCV40_1(X := AI[1,1].Value, Y := AI[1,3].Value);
	AO[1,1].Value := PCV40_1.Y_out;

END_PROGRAM

PROGRAM _EXIT

END_PROGRAM
```

### Program Logical/DCS45_1 (IEC) - Шкаф ШУЭ

#### Variables.var
```iecst
VAR CONSTANT
	def_AI_MC : USINT := 1; (*Количество модулей AI*)
	def_AI_WC : USINT := 4; (*Количество входов в AI*)
	def_AO_MC : USINT := 1; (*Количество модулей AO*)
	def_AO_WC : USINT := 2; (*Количество входов в AO*)
	def_DI_MC : USINT := 4; (*Количество модулей DI*)
	def_DI_WC : USINT := 16; (*Количество входов в DI*)
	def_DO_MC : USINT := 3; (*Количество модулей DO*)
	def_DO_WC : USINT := 16; (*Количество входов в DO*)
END_VAR
VAR
	AI : ARRAY[1..def_AI_MC,1..def_AI_WC] OF FAI;
	AO : ARRAY[1..def_AO_MC,1..def_AO_WC] OF FAO;
	DI : ARRAY[1..def_DI_MC,1..def_DI_WC] OF FDI;
	DO_ : ARRAY[1..def_DO_MC,1..def_DO_WC] OF FDO;
	i : USINT;
	j : USINT;
	KM : ARRAY[1..56] OF FMotor;
END_VAR
```

#### Main.st
```iecst
PROGRAM _INIT

END_PROGRAM

PROGRAM _CYCLIC
	FOR i := 1 TO def_AI_MC DO
		FOR j := 1 TO def_AI_WC DO
			AI[i,j]();
		END_FOR
	END_FOR
	FOR i := 1 TO def_AO_MC DO
		FOR j := 1 TO def_AO_WC DO
			AO[i,j]();
		END_FOR
	END_FOR
	FOR i := 1 TO def_DI_MC DO
		FOR j := 1 TO def_DI_WC DO
			DI[i,j]();
		END_FOR
	END_FOR
	FOR i := 1 TO def_DO_MC DO
		FOR j := 1 TO def_DO_WC DO
			DO_[i,j]();
		END_FOR
	END_FOR
	//KM 1
	KM[1](RunDI := DI[1,3].Out);
	DO_[1,1].In  := KM[1].StopDO;
	DO_[1,2].In  := KM[1].StartDO;
	//KM 2
	KM[2].RunDI := DI[1,4].Out;
	DO_[1,3].In  := KM[2].StopDO;
	DO_[1,4].In  := KM[2].StartDO;
	//KM 3
	KM[3].RunDI := DI[1,5].Out;
	DO_[1,5].In  := KM[3].StopDO;
	DO_[1,6].In  := KM[3].StartDO;
	//KM 4
	KM[4].RunDI := DI[1,6].Out;
	DO_[1,7].In  := KM[4].StopDO;
	DO_[1,8].In  := KM[4].StartDO;
	//KM 5
	KM[5].RunDI := DI[1,7].Out;
	DO_[1,9].In  := KM[5].StopDO;
	DO_[1,10].In  := KM[5].StartDO;
	//KM 6
	KM[6].RunDI := DI[1,8].Out;
	DO_[1,11].In  := KM[6].StopDO;
	DO_[1,12].In  := KM[6].StartDO;
	//KM 7
	KM[7].RunDI := DI[1,9].Out;
	DO_[1,13].In  := KM[7].StopDO;
	DO_[1,14].In  := KM[7].StartDO;
	//KM 8
	KM[8].RunDI := DI[1,10].Out;
	DO_[1,15].In  := KM[8].StopDO;
	DO_[1,16].In  := KM[8].StartDO;
	//KM 9
	KM[9].RunDI := DI[1,11].Out;
	DO_[2,1].In  := KM[9].StopDO;
	DO_[2,2].In  := KM[9].StartDO;
	//KM 10
	KM[10].RunDI := DI[1,12].Out;
	DO_[2,3].In  := KM[10].StopDO;
	DO_[2,4].In  := KM[10].StartDO;
	//KM 11
	KM[11].RunDI := DI[1,13].Out;
	DO_[2,5].In  := KM[11].StopDO;
	DO_[2,6].In  := KM[11].StartDO;
	//KM 12
	KM[12].RunDI := DI[1,14].Out;
	DO_[2,7].In  := KM[12].StopDO;
	DO_[2,8].In  := KM[12].StartDO;
	//KM 13
	KM[13].RunDI := DI[1,15].Out;
	DO_[2,9].In  := KM[13].StopDO;
	DO_[2,10].In  := KM[13].StartDO;
	//KM 14
	KM[14].RunDI := DI[1,16].Out;
	DO_[2,11].In  := KM[14].StopDO;
	DO_[2,12].In  := KM[14].StartDO;
	//KM 15
	KM[15].RunDI := DI[2,1].Out;
	DO_[2,13].In  := KM[15].StopDO;
	DO_[2,14].In  := KM[15].StartDO;
	//KM 16
	KM[16].RunDI := DI[2,2].Out;
	DO_[2,15].In  := KM[16].StopDO;
	DO_[2,16].In  := KM[16].StartDO;
	//KM 17
	KM[17].RunDI := DI[2,3].Out;
	DO_[3,1].In  := KM[17].StopDO;
	DO_[3,2].In  := KM[17].StartDO;
	//KM 18
	KM[18].RunDI := DI[2,4].Out;
	DO_[3,3].In  := KM[18].StopDO;
	DO_[3,4].In  := KM[18].StartDO;

END_PROGRAM

PROGRAM _EXIT

END_PROGRAM
```

Listed in the project but not available here: Logical/Global.typ, Logical/Global.var, Logical/Libraries/Lib489/Constants.var, Logical/Libraries/LibIP001/Constants.var
